LIN {X 0,Y 248.966,Z 382.302,A -85,B 0,C 180,E1 -18796.531,E2 -18796.531} C_VEL
LIN {X 0,Y 248.134,Z 387.569,A -85,B 0,C 180,E1 -18798.563,E2 -18798.563} C_VEL
LIN {X 0,Y 247.427,Z 392.65,A -85,B 0,C 180,E1 -18801.011,E2 -18801.011} C_VEL
LIN {X 0,Y 247.018,Z 396.559,A -85,B 0,C 180,E1 -18803.464,E2 -18803.464} C_VEL
LIN {X 0,Y 246.885,Z 398.563,A -85,B 0,C 180,E1 -18805.099,E2 -18805.099} C_VEL
LIN {X 0,Y 246.837,Z 400.141,A -85,B 0,C 180,E1 -18806.734,E2 -18806.734} C_VEL
LIN {X 0,Y 246.861,Z 401.271,A -85,B 0,C 180,E1 -18808.367,E2 -18808.367} C_VEL
LIN {X 0,Y 246.921,Z 401.968,A -85,B 0,C 180,E1 -18809.998,E2 -18809.998} C_VEL
LIN {X 0,Y 246.86,Z 402.267,A -85,B 0,C 180,E1 -18811.63,E2 -18811.63} C_VEL
LIN {X 0,Y 246.829,Z 402.176,A -85,B 0,C 180,E1 -18813.263,E2 -18813.263} C_VEL
LIN {X 0,Y 246.946,Z 401.583,A -85,B 0,C 180,E1 -18815.062,E2 -18815.062} C_VEL
LIN {X 0,Y 247.394,Z 399.421,A -85,B 0,C 180,E1 -18818.164,E2 -18818.164} C_VEL
LIN {X 0,Y 248.119,Z 396.646,A -85,B 0,C 180,E1 -18820.608,E2 -18820.608} C_VEL
LIN {X 0,Y 249.172,Z 392.86,A -85,B 0,C 180,E1 -18823.039,E2 -18823.039} C_VEL
LIN {X 0,Y 250.607,Z 387.967,A -85,B 0,C 180,E1 -18825.449,E2 -18825.449} C_VEL
LIN {X 0,Y 252.683,Z 381.811,A -85,B 0,C 180,E1 -18827.813,E2 -18827.813} C_VEL
LIN {X 0,Y 254.54,Z 374.922,A -85,B 0,C 180,E1 -18829.967,E2 -18829.967} C_VEL
LIN {X 0,Y 257.036,Z 366.458,A -85,B 0,C 180,E1 -18832.081,E2 -18832.081} C_VEL
LIN {X 0,Y 259.876,Z 355.993,A -85,B 0,C 180,E1 -18834.142,E2 -18834.142} C_VEL
LIN {X 0,Y 262.461,Z 345.405,A -85,B 0,C 180,E1 -18835.791,E2 -18835.791} C_VEL
LIN {X 0,Y 264.624,Z 335.228,A -85,B 0,C 180,E1 -18837.051,E2 -18837.051} C_VEL
LIN {X 0,Y 266.772,Z 323.194,A -85,B 0,C 180,E1 -18838.198,E2 -18838.198} C_VEL
LIN {X 0,Y 268.614,Z 310.075,A -85,B 0,C 180,E1 -18839.108,E2 -18839.108} C_VEL
LIN {X 0,Y 269.834,Z 297.199,A -85,B 0,C 180,E1 -18839.712,E2 -18839.712} C_VEL
LIN {X 0,Y 272.721,Z 239.475,A -85,B 0,C 180,E1 -18841.391,E2 -18841.391} C_VEL
LIN {X 0,Y 270.833,Z 226.518,A -85,B 0,C 180,E1 -18842.191,E2 -18842.191} C_VEL
LIN {X 0,Y 264.34,Z 211.708,A -85,B 0,C 180,E1 -18843.938,E2 -18843.938} C_VEL
LIN {X 0,Y 257.567,Z 198.837,A -85,B 0,C 180,E1 -18845.846,E2 -18845.846} C_VEL
LIN {X 0,Y 254.159,Z 193.208,A -85,B 0,C 180,E1 -18846.839,E2 -18846.839} C_VEL
LIN {X 0,Y 252.073,Z 189.302,A -85,B 0,C 180,E1 -18847.575,E2 -18847.575} C_VEL
LIN {X 0,Y 250.298,Z 183.421,A -85,B 0,C 180,E1 -18850.7,E2 -18850.7} C_VEL
LIN {X 0,Y 249,Z 179.025,A -85,B 0,C 180,E1 -18853.422,E2 -18853.422} C_VEL
LIN {X 0,Y 248.987,Z 178.968,A -85,B 0,C 180,E1 -18857.356,E2 -18857.356} C_VEL
LIN {X 0,Y 249.028,Z 178.958,A -85,B 0,C 180,E1 -18862.201,E2 -18862.201} C_VEL
LIN {X 0,Y 249.035,Z 178.955,A -85,B 0,C 180,E1 -18865.637,E2 -18865.637} C_VEL
LIN {X 0,Y 248.993,Z 178.96,A -85,B 0,C 180,E1 -18869.464,E2 -18869.464} C_VEL
LIN {X 0,Y 249.026,Z 178.955,A -85,B 0,C 180,E1 -18873.156,E2 -18873.156} C_VEL
LIN {X 0,Y 249.042,Z 178.952,A -85,B 0,C 180,E1 -18876.728,E2 -18876.728} C_VEL
LIN {X 0,Y 249.038,Z 178.953,A -85,B 0,C 180,E1 -18880.205,E2 -18880.205} C_VEL
LIN {X 0,Y 249.148,Z 178.944,A -85,B 0,C 180,E1 -18883.615,E2 -18883.615} C_VEL
LIN {X 0,Y 249.177,Z 178.947,A -85,B 0,C 180,E1 -18886.959,E2 -18886.959} C_VEL
LIN {X 0,Y 249.424,Z 178.909,A -85,B 0,C 180,E1 -18891.9,E2 -18891.9} C_VEL
LIN {X 0,Y 249.261,Z 178.934,A -85,B 0,C 180,E1 -18895.147,E2 -18895.147} C_VEL
LIN {X 0,Y 249.647,Z 178.889,A -85,B 0,C 180,E1 -18898.386,E2 -18898.386} C_VEL
LIN {X 0,Y 249.65,Z 178.888,A -85,B 0,C 180,E1 -18901.612,E2 -18901.612} C_VEL
LIN {X 0,Y 249.41,Z 178.911,A -85,B 0,C 180,E1 -18906.758,E2 -18906.758} C_VEL
LIN {X 0,Y 249.322,Z 178.925,A -85,B 0,C 180,E1 -18909.737,E2 -18909.737} C_VEL
LIN {X 0,Y 249.18,Z 178.997,A -85,B 0,C 180,E1 -18913.04,E2 -18913.04} C_VEL
LIN {X 0,Y 250.685,Z 184.007,A -85,B 0,C 180,E1 -18916.071,E2 -18916.071} C_VEL
LIN {X 0,Y 251.242,Z 185.375,A -85,B 0,C 180,E1 -18916.415,E2 -18916.415} C_VEL
LIN {X 0,Y 254.874,Z 191.202,A -85,B 0,C 180,E1 -18917.515,E2 -18917.515} C_VEL
LIN {X 0,Y 259.559,Z 198.978,A -85,B 0,C 180,E1 -18918.864,E2 -18918.864} C_VEL
LIN {X 0,Y 265.571,Z 210.177,A -85,B 0,C 180,E1 -18920.512,E2 -18920.512} C_VEL
LIN {X 0,Y 271.983,Z 224.396,A -85,B 0,C 180,E1 -18922.205,E2 -18922.205} C_VEL
LIN {X 0,Y 273.287,Z 227.948,A -85,B 0,C 180,E1 -18922.557,E2 -18922.557} C_VEL
LIN {X 0,Y 269.932,Z 292.598,A -85,B 0,C 180,E1 -18924.448,E2 -18924.448} C_VEL
LIN {X 0,Y 268.574,Z 306.125,A -85,B 0,C 180,E1 -18925.136,E2 -18925.136} C_VEL
LIN {X 0,Y 266.927,Z 318.251,A -85,B 0,C 180,E1 -18926.045,E2 -18926.045} C_VEL
LIN {X 0,Y 264.797,Z 330.108,A -85,B 0,C 180,E1 -18927.242,E2 -18927.242} C_VEL
LIN {X 0,Y 262.212,Z 342.255,A -85,B 0,C 180,E1 -18928.845,E2 -18928.845} C_VEL
LIN {X 0,Y 259.534,Z 353.022,A -85,B 0,C 180,E1 -18930.689,E2 -18930.689} C_VEL
LIN {X 0,Y 256.751,Z 362.823,A -85,B 0,C 180,E1 -18932.805,E2 -18932.805} C_VEL
LIN {X 0,Y 254.434,Z 370.776,A -85,B 0,C 180,E1 -18934.981,E2 -18934.981} C_VEL
LIN {X 0,Y 252.359,Z 377.241,A -85,B 0,C 180,E1 -18937.177,E2 -18937.177} C_VEL
LIN {X 0,Y 250.679,Z 382.544,A -85,B 0,C 180,E1 -18939.432,E2 -18939.432} C_VEL
LIN {X 0,Y 249.323,Z 386.724,A -85,B 0,C 180,E1 -18941.674,E2 -18941.674} C_VEL
LIN {X 0,Y 247.949,Z 391.02,A -85,B 0,C 180,E1 -18944.881,E2 -18944.881} C_VEL
LIN {X 0,Y 247.175,Z 393.392,A -85,B 0,C 180,E1 -18947.668,E2 -18947.668} C_VEL
LIN {X 0,Y 246.682,Z 394.526,A -85,B 0,C 180,E1 -18950.284,E2 -18950.284} C_VEL
LIN {X 0,Y 246.446,Z 394.592,A -85,B 0,C 180,E1 -18953.214,E2 -18953.214} C_VEL
LIN {X 0,Y 246.423,Z 393.558,A -85,B 0,C 180,E1 -18955.799,E2 -18955.799} C_VEL
LIN {X 0,Y 246.75,Z 391.147,A -85,B 0,C 180,E1 -18958.7,E2 -18958.7} C_VEL
LIN {X 0,Y 247.237,Z 388.115,A -85,B 0,C 180,E1 -18961.105,E2 -18961.105} C_VEL
LIN {X 0,Y 247.938,Z 383.166,A -85,B 0,C 180,E1 -18963.939,E2 -18963.939} C_VEL
LIN {X 0,Y 248.979,Z 376.714,A -85,B 0,C 180,E1 -18966.725,E2 -18966.725} C_VEL
LIN {X 0,Y 250.099,Z 369.969,A -85,B 0,C 180,E1 -18969.007,E2 -18969.007} C_VEL
LIN {X 0,Y 251.742,Z 361.136,A -85,B 0,C 180,E1 -18971.381,E2 -18971.381} C_VEL
LIN {X 0,Y 253.411,Z 351.377,A -85,B 0,C 180,E1 -18973.487,E2 -18973.487} C_VEL
LIN {X 0,Y 254.989,Z 341.933,A -85,B 0,C 180,E1 -18975.121,E2 -18975.121} C_VEL
LIN {X 0,Y 256.718,Z 330.09,A -85,B 0,C 180,E1 -18976.747,E2 -18976.747} C_VEL
LIN {X 0,Y 258.175,Z 318.291,A -85,B 0,C 180,E1 -18978.005,E2 -18978.005} C_VEL
LIN {X 0,Y 259.364,Z 305.706,A -85,B 0,C 180,E1 -18979.002,E2 -18979.002} C_VEL
LIN {X 0,Y 260.44,Z 291.931,A -85,B 0,C 180,E1 -18979.728,E2 -18979.728} C_VEL
LIN {X 0,Y 262.818,Z 221.817,A -85,B 0,C 180,E1 -18981.827,E2 -18981.827} C_VEL
LIN {X 0,Y 261.057,Z 212.59,A -85,B 0,C 180,E1 -18982.293,E2 -18982.293} C_VEL
LIN {X 0,Y 252.445,Z 188.907,A -85,B 0,C 180,E1 -18983.934,E2 -18983.934} C_VEL
LIN {X 0,Y 250.325,Z 183.576,A -85,B 0,C 180,E1 -18984.413,E2 -18984.413} C_VEL
LIN {X 0,Y 249.405,Z 178.982,A -85,B 0,C 180,E1 -18986.367,E2 -18986.367} C_VEL
LIN {X 0,Y 249.674,Z 178.884,A -85,B 0,C 180,E1 -18988.389,E2 -18988.389} C_VEL
LIN {X 0,Y 249.673,Z 178.882,A -85,B 0,C 180,E1 -18991.615,E2 -18991.615} C_VEL
LIN {X 0,Y 249.445,Z 178.912,A -85,B 0,C 180,E1 -18996.472,E2 -18996.472} C_VEL
LIN {X 0,Y 249.341,Z 178.927,A -85,B 0,C 180,E1 -18999.738,E2 -18999.738} C_VEL
LIN {X 0,Y 249.204,Z 178.941,A -85,B 0,C 180,E1 -19004.705,E2 -19004.705} C_VEL
LIN {X 0,Y 249.139,Z 178.942,A -85,B 0,C 180,E1 -19008.079,E2 -19008.079} C_VEL
LIN {X 0,Y 249.087,Z 178.959,A -85,B 0,C 180,E1 -19011.52,E2 -19011.52} C_VEL
LIN {X 0,Y 249.13,Z 178.939,A -85,B 0,C 180,E1 -19015.483,E2 -19015.483} C_VEL
LIN {X 0,Y 249.073,Z 178.955,A -85,B 0,C 180,E1 -19018.99,E2 -19018.99} C_VEL
LIN {X 0,Y 249.031,Z 178.963,A -85,B 0,C 180,E1 -19022.427,E2 -19022.427} C_VEL
LIN {X 0,Y 249.03,Z 178.944,A -85,B 0,C 180,E1 -19026.347,E2 -19026.347} C_VEL
LIN {X 0,Y 249.007,Z 178.965,A -85,B 0,C 180,E1 -19030.479,E2 -19030.479} C_VEL
LIN {X 0,Y 249.008,Z 178.96,A -85,B 0,C 180,E1 -19034.879,E2 -19034.879} C_VEL
LIN {X 0,Y 249.019,Z 178.943,A -85,B 0,C 180,E1 -19037.365,E2 -19037.365} C_VEL
LIN {X 0,Y 249.042,Z 178.955,A -85,B 0,C 180,E1 -19042.202,E2 -19042.202} C_VEL
LIN {X 0,Y 249.044,Z 178.961,A -85,B 0,C 180,E1 -19045.64,E2 -19045.64} C_VEL
LIN {X 0,Y 249.003,Z 178.959,A -85,B 0,C 180,E1 -19049.467,E2 -19049.467} C_VEL
LIN {X 0,Y 249.037,Z 178.962,A -85,B 0,C 180,E1 -19053.159,E2 -19053.159} C_VEL
LIN {X 0,Y 249.059,Z 178.953,A -85,B 0,C 180,E1 -19056.731,E2 -19056.731} C_VEL
LIN {X 0,Y 249.112,Z 178.955,A -85,B 0,C 180,E1 -19060.212,E2 -19060.212} C_VEL
LIN {X 0,Y 249.226,Z 178.935,A -85,B 0,C 180,E1 -19063.622,E2 -19063.622} C_VEL
LIN {X 0,Y 249.246,Z 178.936,A -85,B 0,C 180,E1 -19068.617,E2 -19068.617} C_VEL
LIN {X 0,Y 249.42,Z 178.91,A -85,B 0,C 180,E1 -19071.902,E2 -19071.902} C_VEL
LIN {X 0,Y 249.264,Z 178.933,A -85,B 0,C 180,E1 -19075.149,E2 -19075.149} C_VEL
LIN {X 0,Y 249.663,Z 178.881,A -85,B 0,C 180,E1 -19078.388,E2 -19078.388} C_VEL
LIN {X 0,Y 249.661,Z 178.865,A -85,B 0,C 180,E1 -19081.614,E2 -19081.614} C_VEL
LIN {X 0,Y 249.431,Z 178.906,A -85,B 0,C 180,E1 -19086.472,E2 -19086.472} C_VEL
LIN {X 0,Y 249.347,Z 178.926,A -85,B 0,C 180,E1 -19089.737,E2 -19089.737} C_VEL
LIN {X 0,Y 249.19,Z 178.939,A -85,B 0,C 180,E1 -19092.163,E2 -19092.163} C_VEL
LIN {X 0,Y 248.494,Z 179.024,A -85,B 0,C 180,E1 -19093.513,E2 -19093.513} C_VEL
LIN {X 0,Y 245.601,Z 179.381,A -85,B 0,C 180,E1 -19095.712,E2 -19095.712} C_VEL
LIN {X 0,Y 243.146,Z 179.686,A -85,B 0,C 180,E1 -19097.504,E2 -19097.504} C_VEL
LIN {X 0,Y 242.078,Z 179.824,A -85,B 0,C 180,E1 -19098.895,E2 -19098.895} C_VEL
LIN {X 0,Y 241.982,Z 179.833,A -85,B 0,C 180,E1 -19099.366,E2 -19099.366} C_VEL
LIN {X 0,Y 241.977,Z 179.841,A -85,B 0,C 180,E1 -19102.184,E2 -19102.184} C_VEL
LIN {X 0,Y 241.991,Z 179.824,A -85,B 0,C 180,E1 -19105.827,E2 -19105.827} C_VEL
LIN {X 0,Y 241.972,Z 179.844,A -85,B 0,C 180,E1 -19109.589,E2 -19109.589} C_VEL
LIN {X 0,Y 241.984,Z 179.83,A -85,B 0,C 180,E1 -19113.493,E2 -19113.493} C_VEL
LIN {X 0,Y 241.988,Z 179.841,A -85,B 0,C 180,E1 -19117.583,E2 -19117.583} C_VEL
LIN {X 0,Y 241.912,Z 179.85,A -85,B 0,C 180,E1 -19121.929,E2 -19121.929} C_VEL
LIN {X 0,Y 241.904,Z 179.851,A -85,B 0,C 180,E1 -19126.58,E2 -19126.58} C_VEL
LIN {X 0,Y 241.979,Z 179.842,A -85,B 0,C 180,E1 -19131.646,E2 -19131.646} C_VEL
LIN {X 0,Y 242.01,Z 179.971,A -85,B 0,C 180,E1 -19134.56,E2 -19134.56} C_VEL
LIN {X 0,Y 243.636,Z 187.404,A -85,B 0,C 180,E1 -19137.746,E2 -19137.746} C_VEL
LIN {X 0,Y 244.356,Z 190.774,A -85,B 0,C 180,E1 -19139.014,E2 -19139.014} C_VEL
LIN {X 0,Y 251.771,Z 210.686,A -85,B 0,C 180,E1 -19140.527,E2 -19140.527} C_VEL
LIN {X 0,Y 252.89,Z 215.079,A -85,B 0,C 180,E1 -19140.788,E2 -19140.788} C_VEL
LIN {X 0,Y 256.022,Z 236.939,A -85,B 0,C 180,E1 -19141.825,E2 -19141.825} C_VEL
LIN {X 0,Y 253.703,Z 299.6,A -85,B 0,C 180,E1 -19143.744,E2 -19143.744} C_VEL
LIN {X 0,Y 252.659,Z 312.872,A -85,B 0,C 180,E1 -19144.458,E2 -19144.458} C_VEL
LIN {X 0,Y 251.367,Z 325.12,A -85,B 0,C 180,E1 -19145.423,E2 -19145.423} C_VEL
LIN {X 0,Y 249.605,Z 337.75,A -85,B 0,C 180,E1 -19146.783,E2 -19146.783} C_VEL
LIN {X 0,Y 247.858,Z 349.062,A -85,B 0,C 180,E1 -19148.368,E2 -19148.368} C_VEL
LIN {X 0,Y 246.028,Z 359.736,A -85,B 0,C 180,E1 -19150.275,E2 -19150.275} C_VEL
LIN {X 0,Y 244.414,Z 369.293,A -85,B 0,C 180,E1 -19152.425,E2 -19152.425} C_VEL
LIN {X 0,Y 242.72,Z 378.086,A -85,B 0,C 180,E1 -19154.893,E2 -19154.893} C_VEL
LIN {X 0,Y 241.446,Z 385.083,A -85,B 0,C 180,E1 -19157.389,E2 -19157.389} C_VEL
LIN {X 0,Y 240.614,Z 390.675,A -85,B 0,C 180,E1 -19159.905,E2 -19159.905} C_VEL
LIN {X 0,Y 240.056,Z 395.032,A -85,B 0,C 180,E1 -19162.428,E2 -19162.428} C_VEL
LIN {X 0,Y 239.772,Z 398.622,A -85,B 0,C 180,E1 -19165.269,E2 -19165.269} C_VEL
LIN {X 0,Y 239.775,Z 401.079,A -85,B 0,C 180,E1 -19168.319,E2 -19168.319} C_VEL
LIN {X 0,Y 239.832,Z 401.81,A -85,B 0,C 180,E1 -19169.998,E2 -19169.998} C_VEL
LIN {X 0,Y 239.774,Z 402.14,A -85,B 0,C 180,E1 -19171.678,E2 -19171.678} C_VEL
LIN {X 0,Y 239.846,Z 401.628,A -85,B 0,C 180,E1 -19175.041,E2 -19175.041} C_VEL
LIN {X 0,Y 240.036,Z 400.739,A -85,B 0,C 180,E1 -19176.724,E2 -19176.724} C_VEL
LIN {X 0,Y 240.814,Z 397.763,A -85,B 0,C 180,E1 -19180.083,E2 -19180.083} C_VEL
LIN {X 0,Y 241.82,Z 394.384,A -85,B 0,C 180,E1 -19182.588,E2 -19182.588} C_VEL
LIN {X 0,Y 243.15,Z 389.945,A -85,B 0,C 180,E1 -19185.076,E2 -19185.076} C_VEL
LIN {X 0,Y 245.541,Z 383.27,A -85,B 0,C 180,E1 -19187.918,E2 -19187.918} C_VEL
LIN {X 0,Y 247.416,Z 377.362,A -85,B 0,C 180,E1 -19189.928,E2 -19189.928} C_VEL
LIN {X 0,Y 249.531,Z 370.286,A -85,B 0,C 180,E1 -19191.91,E2 -19191.91} C_VEL
LIN {X 0,Y 252.064,Z 361.749,A -85,B 0,C 180,E1 -19193.844,E2 -19193.844} C_VEL
LIN {X 0,Y 254.899,Z 351.279,A -85,B 0,C 180,E1 -19195.736,E2 -19195.736} C_VEL
LIN {X 0,Y 257.702,Z 339.544,A -85,B 0,C 180,E1 -19197.398,E2 -19197.398} C_VEL
LIN {X 0,Y 260.125,Z 327.788,A -85,B 0,C 180,E1 -19198.655,E2 -19198.655} C_VEL
LIN {X 0,Y 262.049,Z 315.767,A -85,B 0,C 180,E1 -19199.633,E2 -19199.633} C_VEL
LIN {X 0,Y 263.622,Z 302.876,A -85,B 0,C 180,E1 -19200.375,E2 -19200.375} C_VEL
LIN {X 0,Y 264.711,Z 288.127,A -85,B 0,C 180,E1 -19200.888,E2 -19200.888} C_VEL
LIN {X 0,Y 267.122,Z 240.371,A -85,B 0,C 180,E1 -19202.305,E2 -19202.305} C_VEL
LIN {X 0,Y 265.472,Z 229.249,A -85,B 0,C 180,E1 -19203.032,E2 -19203.032} C_VEL
LIN {X 0,Y 259.41,Z 215.401,A -85,B 0,C 180,E1 -19204.745,E2 -19204.745} C_VEL
LIN {X 0,Y 253.533,Z 203.887,A -85,B 0,C 180,E1 -19206.496,E2 -19206.496} C_VEL
LIN {X 0,Y 247.411,Z 193.745,A -85,B 0,C 180,E1 -19208.387,E2 -19208.387} C_VEL
LIN {X 0,Y 244.751,Z 189.183,A -85,B 0,C 180,E1 -19209.374,E2 -19209.374} C_VEL
LIN {X 0,Y 242.894,Z 183.212,A -85,B 0,C 180,E1 -19212.841,E2 -19212.841} C_VEL
LIN {X 0,Y 241.914,Z 179.884,A -85,B 0,C 180,E1 -19215.144,E2 -19215.144} C_VEL
LIN {X 0,Y 241.905,Z 179.847,A -85,B 0,C 180,E1 -19219.054,E2 -19219.054} C_VEL
LIN {X 0,Y 241.974,Z 179.836,A -85,B 0,C 180,E1 -19222.414,E2 -19222.414} C_VEL
LIN {X 0,Y 241.972,Z 179.838,A -85,B 0,C 180,E1 -19226.505,E2 -19226.505} C_VEL
LIN {X 0,Y 241.968,Z 179.844,A -85,B 0,C 180,E1 -19230.611,E2 -19230.611} C_VEL
LIN {X 0,Y 242.024,Z 179.835,A -85,B 0,C 180,E1 -19234.177,E2 -19234.177} C_VEL
LIN {X 0,Y 241.983,Z 179.841,A -85,B 0,C 180,E1 -19238.332,E2 -19238.332} C_VEL
LIN {X 0,Y 242.104,Z 179.824,A -85,B 0,C 180,E1 -19243.317,E2 -19243.317} C_VEL
LIN {X 0,Y 242.151,Z 179.812,A -85,B 0,C 180,E1 -19248.277,E2 -19248.277} C_VEL
LIN {X 0,Y 242.373,Z 179.789,A -85,B 0,C 180,E1 -19251.663,E2 -19251.663} C_VEL
LIN {X 0,Y 242.395,Z 179.781,A -85,B 0,C 180,E1 -19253.339,E2 -19253.339} C_VEL
LIN {X 0,Y 242.607,Z 179.765,A -85,B 0,C 180,E1 -19258.339,E2 -19258.339} C_VEL
LIN {X 0,Y 242.609,Z 179.765,A -85,B 0,C 180,E1 -19261.659,E2 -19261.659} C_VEL
LIN {X 0,Y 242.39,Z 179.786,A -85,B 0,C 180,E1 -19266.731,E2 -19266.731} C_VEL
LIN {X 0,Y 242.25,Z 179.808,A -85,B 0,C 180,E1 -19270.024,E2 -19270.024} C_VEL
LIN {X 0,Y 242.187,Z 179.963,A -85,B 0,C 180,E1 -19271.507,E2 -19271.507} C_VEL
LIN {X 0,Y 243.558,Z 184.504,A -85,B 0,C 180,E1 -19274.357,E2 -19274.357} C_VEL
LIN {X 0,Y 246.527,Z 189.136,A -85,B 0,C 180,E1 -19275.448,E2 -19275.448} C_VEL
LIN {X 0,Y 253.165,Z 199.962,A -85,B 0,C 180,E1 -19277.531,E2 -19277.531} C_VEL
LIN {X 0,Y 260.169,Z 212.884,A -85,B 0,C 180,E1 -19279.585,E2 -19279.585} C_VEL
LIN {X 0,Y 266,Z 225.762,A -85,B 0,C 180,E1 -19281.205,E2 -19281.205} C_VEL
LIN {X 0,Y 267.675,Z 229.833,A -85,B 0,C 180,E1 -19281.664,E2 -19281.664} C_VEL
LIN {X 0,Y 264.236,Z 292.445,A -85,B 0,C 180,E1 -19283.535,E2 -19283.535} C_VEL
LIN {X 0,Y 262.797,Z 306.223,A -85,B 0,C 180,E1 -19284.246,E2 -19284.246} C_VEL
LIN {X 0,Y 260.891,Z 319.326,A -85,B 0,C 180,E1 -19285.26,E2 -19285.26} C_VEL
LIN {X 0,Y 258.537,Z 331.741,A -85,B 0,C 180,E1 -19286.568,E2 -19286.568} C_VEL
LIN {X 0,Y 255.948,Z 343.152,A -85,B 0,C 180,E1 -19288.139,E2 -19288.139} C_VEL
LIN {X 0,Y 253.205,Z 353.544,A -85,B 0,C 180,E1 -19289.973,E2 -19289.973} C_VEL
LIN {X 0,Y 250.587,Z 362.306,A -85,B 0,C 180,E1 -19291.898,E2 -19291.898} C_VEL
LIN {X 0,Y 248.165,Z 370.229,A -85,B 0,C 180,E1 -19294.076,E2 -19294.076} C_VEL
LIN {X 0,Y 245.558,Z 377.876,A -85,B 0,C 180,E1 -19296.743,E2 -19296.743} C_VEL
LIN {X 0,Y 243.545,Z 383.746,A -85,B 0,C 180,E1 -19299.408,E2 -19299.408} C_VEL
LIN {X 0,Y 242.081,Z 387.942,A -85,B 0,C 180,E1 -19301.891,E2 -19301.891} C_VEL
LIN {X 0,Y 241.018,Z 391.097,A -85,B 0,C 180,E1 -19304.412,E2 -19304.412} C_VEL
LIN {X 0,Y 240.075,Z 393.741,A -85,B 0,C 180,E1 -19307.68,E2 -19307.68} C_VEL
LIN {X 0,Y 239.641,Z 394.59,A -85,B 0,C 180,E1 -19309.823,E2 -19309.823} C_VEL
LIN {X 0,Y 239.375,Z 394.773,A -85,B 0,C 180,E1 -19312.439,E2 -19312.439} C_VEL
LIN {X 0,Y 239.303,Z 393.855,A -85,B 0,C 180,E1 -19315.316,E2 -19315.316} C_VEL
LIN {X 0,Y 239.586,Z 391.661,A -85,B 0,C 180,E1 -19318.285,E2 -19318.285} C_VEL
LIN {X 0,Y 240.199,Z 387.896,A -85,B 0,C 180,E1 -19321.373,E2 -19321.373} C_VEL
LIN {X 0,Y 240.872,Z 383.325,A -85,B 0,C 180,E1 -19324.048,E2 -19324.048} C_VEL
LIN {X 0,Y 241.95,Z 376.884,A -85,B 0,C 180,E1 -19326.915,E2 -19326.915} C_VEL
LIN {X 0,Y 243.088,Z 370.164,A -85,B 0,C 180,E1 -19329.26,E2 -19329.26} C_VEL
LIN {X 0,Y 244.707,Z 361.812,A -85,B 0,C 180,E1 -19331.586,E2 -19331.586} C_VEL
LIN {X 0,Y 246.477,Z 351.827,A -85,B 0,C 180,E1 -19333.818,E2 -19333.818} C_VEL
LIN {X 0,Y 248.289,Z 341.402,A -85,B 0,C 180,E1 -19335.662,E2 -19335.662} C_VEL
LIN {X 0,Y 250.109,Z 329.213,A -85,B 0,C 180,E1 -19337.353,E2 -19337.353} C_VEL
LIN {X 0,Y 251.546,Z 317.754,A -85,B 0,C 180,E1 -19338.583,E2 -19338.583} C_VEL
LIN {X 0,Y 252.786,Z 304.681,A -85,B 0,C 180,E1 -19339.616,E2 -19339.616} C_VEL
LIN {X 0,Y 253.893,Z 290.762,A -85,B 0,C 180,E1 -19340.341,E2 -19340.341} C_VEL
LIN {X 0,Y 256.246,Z 222.797,A -85,B 0,C 180,E1 -19342.413,E2 -19342.413} C_VEL
LIN {X 0,Y 254.735,Z 214.758,A -85,B 0,C 180,E1 -19342.828,E2 -19342.828} C_VEL
LIN {X 0,Y 246.327,Z 191.636,A -85,B 0,C 180,E1 -19344.487,E2 -19344.487} C_VEL
LIN {X 0,Y 243.215,Z 184.115,A -85,B 0,C 180,E1 -19345.133,E2 -19345.133} C_VEL
LIN {X 0,Y 242.951,Z 183.003,A -85,B 0,C 180,E1 -19345.439,E2 -19345.439} C_VEL
LIN {X 0,Y 242.41,Z 179.845,A -85,B 0,C 180,E1 -19346.886,E2 -19346.886} C_VEL
LIN {X 0,Y 242.689,Z 179.752,A -85,B 0,C 180,E1 -19350.002,E2 -19350.002} C_VEL
LIN {X 0,Y 242.633,Z 179.759,A -85,B 0,C 180,E1 -19351.662,E2 -19351.662} C_VEL
LIN {X 0,Y 242.415,Z 179.788,A -85,B 0,C 180,E1 -19356.661,E2 -19356.661} C_VEL
LIN {X 0,Y 242.265,Z 179.808,A -85,B 0,C 180,E1 -19360.025,E2 -19360.025} C_VEL
LIN {X 0,Y 242.166,Z 179.819,A -85,B 0,C 180,E1 -19365.142,E2 -19365.142} C_VEL
LIN {X 0,Y 242.073,Z 179.82,A -85,B 0,C 180,E1 -19368.626,E2 -19368.626} C_VEL
LIN {X 0,Y 242.013,Z 179.838,A -85,B 0,C 180,E1 -19372.181,E2 -19372.181} C_VEL
LIN {X 0,Y 242.067,Z 179.817,A -85,B 0,C 180,E1 -19375.84,E2 -19375.84} C_VEL
LIN {X 0,Y 242.007,Z 179.839,A -85,B 0,C 180,E1 -19379.585,E2 -19379.585} C_VEL
LIN {X 0,Y 241.981,Z 179.835,A -85,B 0,C 180,E1 -19383.494,E2 -19383.494} C_VEL
LIN {X 0,Y 241.986,Z 179.827,A -85,B 0,C 180,E1 -19387.584,E2 -19387.584} C_VEL
LIN {X 0,Y 241.94,Z 179.846,A -85,B 0,C 180,E1 -19391.923,E2 -19391.923} C_VEL
LIN {X 0,Y 241.938,Z 179.829,A -85,B 0,C 180,E1 -19396.572,E2 -19396.572} C_VEL
LIN {X 0,Y 241.957,Z 179.825,A -85,B 0,C 180,E1 -19400.282,E2 -19400.282} C_VEL
LIN {X 0,Y 241.981,Z 179.843,A -85,B 0,C 180,E1 -19404.489,E2 -19404.489} C_VEL
LIN {X 0,Y 241.954,Z 179.84,A -85,B 0,C 180,E1 -19408.478,E2 -19408.478} C_VEL
LIN {X 0,Y 241.97,Z 179.845,A -85,B 0,C 180,E1 -19412.309,E2 -19412.309} C_VEL
LIN {X 0,Y 242.028,Z 179.831,A -85,B 0,C 180,E1 -19416.014,E2 -19416.014} C_VEL
LIN {X 0,Y 242.039,Z 179.832,A -85,B 0,C 180,E1 -19419.609,E2 -19419.609} C_VEL
LIN {X 0,Y 242.167,Z 179.814,A -85,B 0,C 180,E1 -19423.279,E2 -19423.279} C_VEL
LIN {X 0,Y 242.182,Z 179.817,A -85,B 0,C 180,E1 -19428.28,E2 -19428.28} C_VEL
LIN {X 0,Y 242.374,Z 179.788,A -85,B 0,C 180,E1 -19431.665,E2 -19431.665} C_VEL
LIN {X 0,Y 242.399,Z 179.783,A -85,B 0,C 180,E1 -19433.341,E2 -19433.341} C_VEL
LIN {X 0,Y 242.622,Z 179.758,A -85,B 0,C 180,E1 -19438.341,E2 -19438.341} C_VEL
LIN {X 0,Y 242.621,Z 179.74,A -85,B 0,C 180,E1 -19441.661,E2 -19441.661} C_VEL
LIN {X 0,Y 242.404,Z 179.781,A -85,B 0,C 180,E1 -19446.66,E2 -19446.66} C_VEL
LIN {X 0,Y 242.27,Z 179.806,A -85,B 0,C 180,E1 -19450.024,E2 -19450.024} C_VEL
LIN {X 0,Y 242.125,Z 179.804,A -85,B 0,C 180,E1 -19455.144,E2 -19455.144} C_VEL
LIN {X 0,Y 241.982,Z 179.833,A -85,B 0,C 180,E1 -19459.366,E2 -19459.366} C_VEL
LIN {X 0,Y 241.308,Z 179.927,A -85,B 0,C 180,E1 -19460.754,E2 -19460.754} C_VEL
LIN {X 0,Y 238.507,Z 180.273,A -85,B 0,C 180,E1 -19463.019,E2 -19463.019} C_VEL
LIN {X 0,Y 235.282,Z 180.663,A -85,B 0,C 180,E1 -19465.812,E2 -19465.812} C_VEL
LIN {X 0,Y 234.92,Z 180.705,A -85,B 0,C 180,E1 -19466.778,E2 -19466.778} C_VEL
LIN {X 0,Y 234.903,Z 180.725,A -85,B 0,C 180,E1 -19470.573,E2 -19470.573} C_VEL
LIN {X 0,Y 234.93,Z 180.709,A -85,B 0,C 180,E1 -19474.639,E2 -19474.639} C_VEL
LIN {X 0,Y 234.917,Z 180.716,A -85,B 0,C 180,E1 -19478.935,E2 -19478.935} C_VEL
LIN {X 0,Y 234.858,Z 180.728,A -85,B 0,C 180,E1 -19483.494,E2 -19483.494} C_VEL
LIN {X 0,Y 234.856,Z 180.728,A -85,B 0,C 180,E1 -19486.505,E2 -19486.505} C_VEL
LIN {X 0,Y 234.923,Z 180.72,A -85,B 0,C 180,E1 -19491.078,E2 -19491.078} C_VEL
LIN {X 0,Y 234.94,Z 180.887,A -85,B 0,C 180,E1 -19494.03,E2 -19494.03} C_VEL
LIN {X 0,Y 236.795,Z 189.252,A -85,B 0,C 180,E1 -19497.706,E2 -19497.706} C_VEL
LIN {X 0,Y 237.088,Z 190.758,A -85,B 0,C 180,E1 -19498.19,E2 -19498.19} C_VEL
LIN {X 0,Y 243.253,Z 206.795,A -85,B 0,C 180,E1 -19499.511,E2 -19499.511} C_VEL
LIN {X 0,Y 246.356,Z 215.976,A -85,B 0,C 180,E1 -19500.162,E2 -19500.162} C_VEL
LIN {X 0,Y 249.461,Z 238.081,A -85,B 0,C 180,E1 -19501.242,E2 -19501.242} C_VEL
LIN {X 0,Y 247.076,Z 299.144,A -85,B 0,C 180,E1 -19503.155,E2 -19503.155} C_VEL
LIN {X 0,Y 245.941,Z 313.266,A -85,B 0,C 180,E1 -19503.936,E2 -19503.936} C_VEL
LIN {X 0,Y 244.619,Z 325.356,A -85,B 0,C 180,E1 -19504.926,E2 -19504.926} C_VEL
LIN {X 0,Y 242.814,Z 337.91,A -85,B 0,C 180,E1 -19506.32,E2 -19506.32} C_VEL
LIN {X 0,Y 241.009,Z 349.174,A -85,B 0,C 180,E1 -19507.947,E2 -19507.947} C_VEL
LIN {X 0,Y 239.252,Z 359.079,A -85,B 0,C 180,E1 -19509.754,E2 -19509.754} C_VEL
LIN {X 0,Y 237.614,Z 368.5,A -85,B 0,C 180,E1 -19511.905,E2 -19511.905} C_VEL
LIN {X 0,Y 235.851,Z 377.436,A -85,B 0,C 180,E1 -19514.442,E2 -19514.442} C_VEL
LIN {X 0,Y 234.46,Z 384.55,A -85,B 0,C 180,E1 -19517.006,E2 -19517.006} C_VEL
LIN {X 0,Y 233.585,Z 390.229,A -85,B 0,C 180,E1 -19519.598,E2 -19519.598} C_VEL
LIN {X 0,Y 233.01,Z 394.666,A -85,B 0,C 180,E1 -19522.198,E2 -19522.198} C_VEL
LIN {X 0,Y 232.677,Z 398.613,A -85,B 0,C 180,E1 -19525.397,E2 -19525.397} C_VEL
LIN {X 0,Y 232.672,Z 400.863,A -85,B 0,C 180,E1 -19528.267,E2 -19528.267} C_VEL
LIN {X 0,Y 232.745,Z 401.65,A -85,B 0,C 180,E1 -19529.998,E2 -19529.998} C_VEL
LIN {X 0,Y 232.67,Z 402.012,A -85,B 0,C 180,E1 -19531.729,E2 -19531.729} C_VEL
LIN {X 0,Y 232.77,Z 401.57,A -85,B 0,C 180,E1 -19535.195,E2 -19535.195} C_VEL
LIN {X 0,Y 232.982,Z 400.738,A -85,B 0,C 180,E1 -19536.928,E2 -19536.928} C_VEL
LIN {X 0,Y 233.806,Z 397.829,A -85,B 0,C 180,E1 -19540.388,E2 -19540.388} C_VEL
LIN {X 0,Y 234.877,Z 394.532,A -85,B 0,C 180,E1 -19542.966,E2 -19542.966} C_VEL
LIN {X 0,Y 236.298,Z 390.186,A -85,B 0,C 180,E1 -19545.524,E2 -19545.524} C_VEL
LIN {X 0,Y 238.819,Z 383.637,A -85,B 0,C 180,E1 -19548.44,E2 -19548.44} C_VEL
LIN {X 0,Y 240.74,Z 377.797,A -85,B 0,C 180,E1 -19550.505,E2 -19550.505} C_VEL
LIN {X 0,Y 243.473,Z 369.264,A -85,B 0,C 180,E1 -19552.933,E2 -19552.933} C_VEL
LIN {X 0,Y 246.198,Z 360.53,A -85,B 0,C 180,E1 -19554.899,E2 -19554.899} C_VEL
LIN {X 0,Y 249.195,Z 349.868,A -85,B 0,C 180,E1 -19556.821,E2 -19556.821} C_VEL
LIN {X 0,Y 251.856,Z 339.292,A -85,B 0,C 180,E1 -19558.317,E2 -19558.317} C_VEL
LIN {X 0,Y 254.353,Z 327.556,A -85,B 0,C 180,E1 -19559.595,E2 -19559.595} C_VEL
LIN {X 0,Y 256.591,Z 314.303,A -85,B 0,C 180,E1 -19560.67,E2 -19560.67} C_VEL
LIN {X 0,Y 258.138,Z 301.125,A -85,B 0,C 180,E1 -19561.404,E2 -19561.404} C_VEL
LIN {X 0,Y 259.436,Z 282.027,A -85,B 0,C 180,E1 -19562.034,E2 -19562.034} C_VEL
LIN {X 0,Y 261.613,Z 241.358,A -85,B 0,C 180,E1 -19563.257,E2 -19563.257} C_VEL
LIN {X 0,Y 260.1,Z 231.705,A -85,B 0,C 180,E1 -19563.933,E2 -19563.933} C_VEL
LIN {X 0,Y 254.564,Z 219.061,A -85,B 0,C 180,E1 -19565.596,E2 -19565.596} C_VEL
LIN {X 0,Y 249.089,Z 208.286,A -85,B 0,C 180,E1 -19567.299,E2 -19567.299} C_VEL
LIN {X 0,Y 243.374,Z 198.558,A -85,B 0,C 180,E1 -19569.187,E2 -19569.187} C_VEL
LIN {X 0,Y 240.376,Z 193.825,A -85,B 0,C 180,E1 -19570.237,E2 -19570.237} C_VEL
LIN {X 0,Y 237.566,Z 189.321,A -85,B 0,C 180,E1 -19571.329,E2 -19571.329} C_VEL
LIN {X 0,Y 236.988,Z 187.699,A -85,B 0,C 180,E1 -19572.149,E2 -19572.149} C_VEL
LIN {X 0,Y 234.972,Z 181.275,A -85,B 0,C 180,E1 -19576.533,E2 -19576.533} C_VEL
LIN {X 0,Y 234.848,Z 180.731,A -85,B 0,C 180,E1 -19577.284,E2 -19577.284} C_VEL
LIN {X 0,Y 234.911,Z 180.723,A -85,B 0,C 180,E1 -19581.076,E2 -19581.076} C_VEL
LIN {X 0,Y 234.921,Z 180.713,A -85,B 0,C 180,E1 -19585.36,E2 -19585.36} C_VEL
LIN {X 0,Y 234.89,Z 180.716,A -85,B 0,C 180,E1 -19589.425,E2 -19589.425} C_VEL
LIN {X 0,Y 234.96,Z 180.711,A -85,B 0,C 180,E1 -19593.805,E2 -19593.805} C_VEL
LIN {X 0,Y 234.956,Z 180.712,A -85,B 0,C 180,E1 -19598.006,E2 -19598.006} C_VEL
LIN {X 0,Y 235.045,Z 180.705,A -85,B 0,C 180,E1 -19603.092,E2 -19603.092} C_VEL
LIN {X 0,Y 235.084,Z 180.694,A -85,B 0,C 180,E1 -19607.92,E2 -19607.92} C_VEL
LIN {X 0,Y 235.307,Z 180.672,A -85,B 0,C 180,E1 -19611.411,E2 -19611.411} C_VEL
LIN {X 0,Y 235.346,Z 180.658,A -85,B 0,C 180,E1 -19613.139,E2 -19613.139} C_VEL
LIN {X 0,Y 235.567,Z 180.642,A -85,B 0,C 180,E1 -19618.29,E2 -19618.29} C_VEL
LIN {X 0,Y 235.568,Z 180.643,A -85,B 0,C 180,E1 -19621.709,E2 -19621.709} C_VEL
LIN {X 0,Y 235.347,Z 180.664,A -85,B 0,C 180,E1 -19626.86,E2 -19626.86} C_VEL
LIN {X 0,Y 235.288,Z 180.898,A -85,B 0,C 180,E1 -19629.717,E2 -19629.717} C_VEL
LIN {X 0,Y 236.398,Z 184.856,A -85,B 0,C 180,E1 -19632.337,E2 -19632.337} C_VEL
LIN {X 0,Y 239.346,Z 189.356,A -85,B 0,C 180,E1 -19633.526,E2 -19633.526} C_VEL
LIN {X 0,Y 243.681,Z 195.883,A -85,B 0,C 180,E1 -19635.044,E2 -19635.044} C_VEL
LIN {X 0,Y 249.372,Z 205.479,A -85,B 0,C 180,E1 -19636.923,E2 -19636.923} C_VEL
LIN {X 0,Y 255.603,Z 217.046,A -85,B 0,C 180,E1 -19638.819,E2 -19638.819} C_VEL
LIN {X 0,Y 261.095,Z 229.541,A -85,B 0,C 180,E1 -19640.451,E2 -19640.451} C_VEL
LIN {X 0,Y 262.115,Z 231.983,A -85,B 0,C 180,E1 -19640.74,E2 -19640.74} C_VEL
LIN {X 0,Y 258.653,Z 292.451,A -85,B 0,C 180,E1 -19642.577,E2 -19642.577} C_VEL
LIN {X 0,Y 257.139,Z 306.152,A -85,B 0,C 180,E1 -19643.286,E2 -19643.286} C_VEL
LIN {X 0,Y 255.275,Z 318.822,A -85,B 0,C 180,E1 -19644.276,E2 -19644.276} C_VEL
LIN {X 0,Y 252.776,Z 331.342,A -85,B 0,C 180,E1 -19645.601,E2 -19645.601} C_VEL
LIN {X 0,Y 250.311,Z 341.886,A -85,B 0,C 180,E1 -19647.054,E2 -19647.054} C_VEL
LIN {X 0,Y 247.429,Z 352.344,A -85,B 0,C 180,E1 -19648.872,E2 -19648.872} C_VEL
LIN {X 0,Y 244.475,Z 361.92,A -85,B 0,C 180,E1 -19650.981,E2 -19650.981} C_VEL
LIN {X 0,Y 241.841,Z 370.063,A -85,B 0,C 180,E1 -19653.243,E2 -19653.243} C_VEL
LIN {X 0,Y 239.005,Z 377.91,A -85,B 0,C 180,E1 -19656.022,E2 -19656.022} C_VEL
LIN {X 0,Y 237.056,Z 383.319,A -85,B 0,C 180,E1 -19658.504,E2 -19658.504} C_VEL
LIN {X 0,Y 235.081,Z 388.482,A -85,B 0,C 180,E1 -19661.638,E2 -19661.638} C_VEL
LIN {X 0,Y 234.096,Z 391.173,A -85,B 0,C 180,E1 -19663.906,E2 -19663.906} C_VEL
LIN {X 0,Y 233.333,Z 393.207,A -85,B 0,C 180,E1 -19666.292,E2 -19666.292} C_VEL
LIN {X 0,Y 232.688,Z 394.574,A -85,B 0,C 180,E1 -19669.032,E2 -19669.032} C_VEL
LIN {X 0,Y 232.308,Z 394.924,A -85,B 0,C 180,E1 -19671.865,E2 -19671.865} C_VEL
LIN {X 0,Y 232.187,Z 394.105,A -85,B 0,C 180,E1 -19674.896,E2 -19674.896} C_VEL
LIN {X 0,Y 232.413,Z 392.107,A -85,B 0,C 180,E1 -19677.853,E2 -19677.853} C_VEL
LIN {X 0,Y 233.054,Z 388.4,A -85,B 0,C 180,E1 -19681.154,E2 -19681.154} C_VEL
LIN {X 0,Y 233.854,Z 383.075,A -85,B 0,C 180,E1 -19684.366,E2 -19684.366} C_VEL
LIN {X 0,Y 234.899,Z 377.03,A -85,B 0,C 180,E1 -19687.113,E2 -19687.113} C_VEL
LIN {X 0,Y 236.092,Z 370.312,A -85,B 0,C 180,E1 -19689.529,E2 -19689.529} C_VEL
LIN {X 0,Y 237.771,Z 361.932,A -85,B 0,C 180,E1 -19691.929,E2 -19691.929} C_VEL
LIN {X 0,Y 239.412,Z 352.882,A -85,B 0,C 180,E1 -19694.028,E2 -19694.028} C_VEL
LIN {X 0,Y 241.221,Z 342.97,A -85,B 0,C 180,E1 -19695.879,E2 -19695.879} C_VEL
LIN {X 0,Y 242.892,Z 332.355,A -85,B 0,C 180,E1 -19697.469,E2 -19697.469} C_VEL
LIN {X 0,Y 244.632,Z 319.717,A -85,B 0,C 180,E1 -19698.925,E2 -19698.925} C_VEL
LIN {X 0,Y 245.952,Z 306.952,A -85,B 0,C 180,E1 -19700.026,E2 -19700.026} C_VEL
LIN {X 0,Y 247.051,Z 293.627,A -85,B 0,C 180,E1 -19700.794,E2 -19700.794} C_VEL
LIN {X 0,Y 247.998,Z 272.807,A -85,B 0,C 180,E1 -19701.497,E2 -19701.497} C_VEL
LIN {X 0,Y 249.721,Z 223.936,A -85,B 0,C 180,E1 -19703.007,E2 -19703.007} C_VEL
LIN {X 0,Y 248.485,Z 217.167,A -85,B 0,C 180,E1 -19703.365,E2 -19703.365} C_VEL
LIN {X 0,Y 240.43,Z 194.935,A -85,B 0,C 180,E1 -19705.013,E2 -19705.013} C_VEL
LIN {X 0,Y 235.982,Z 184.077,A -85,B 0,C 180,E1 -19705.97,E2 -19705.97} C_VEL
LIN {X 0,Y 235.448,Z 180.977,A -85,B 0,C 180,E1 -19707.222,E2 -19707.222} C_VEL
LIN {X 0,Y 235.516,Z 180.649,A -85,B 0,C 180,E1 -19707.864,E2 -19707.864} C_VEL
LIN {X 0,Y 235.653,Z 180.628,A -85,B 0,C 180,E1 -19710.002,E2 -19710.002} C_VEL
LIN {X 0,Y 235.593,Z 180.636,A -85,B 0,C 180,E1 -19711.711,E2 -19711.711} C_VEL
LIN {X 0,Y 235.366,Z 180.666,A -85,B 0,C 180,E1 -19716.861,E2 -19716.861} C_VEL
LIN {X 0,Y 235.211,Z 180.686,A -85,B 0,C 180,E1 -19720.329,E2 -19720.329} C_VEL
LIN {X 0,Y 235.113,Z 180.7,A -85,B 0,C 180,E1 -19725.608,E2 -19725.608} C_VEL
LIN {X 0,Y 235.009,Z 180.699,A -85,B 0,C 180,E1 -19729.207,E2 -19729.207} C_VEL
LIN {X 0,Y 234.961,Z 180.718,A -85,B 0,C 180,E1 -19732.884,E2 -19732.884} C_VEL
LIN {X 0,Y 234.968,Z 180.699,A -85,B 0,C 180,E1 -19736.659,E2 -19736.659} C_VEL
LIN {X 0,Y 234.923,Z 180.721,A -85,B 0,C 180,E1 -19740.571,E2 -19740.571} C_VEL
LIN {X 0,Y 234.927,Z 180.706,A -85,B 0,C 180,E1 -19744.64,E2 -19744.64} C_VEL
LIN {X 0,Y 234.943,Z 180.71,A -85,B 0,C 180,E1 -19748.946,E2 -19748.946} C_VEL
LIN {X 0,Y 234.891,Z 180.722,A -85,B 0,C 180,E1 -19753.487,E2 -19753.487} C_VEL
LIN {X 0,Y 234.891,Z 180.705,A -85,B 0,C 180,E1 -19756.516,E2 -19756.516} C_VEL
LIN {X 0,Y 234.919,Z 180.708,A -85,B 0,C 180,E1 -19761.08,E2 -19761.08} C_VEL
LIN {X 0,Y 234.927,Z 180.72,A -85,B 0,C 180,E1 -19765.362,E2 -19765.362} C_VEL
LIN {X 0,Y 234.901,Z 180.715,A -85,B 0,C 180,E1 -19769.429,E2 -19769.429} C_VEL
LIN {X 0,Y 234.971,Z 180.715,A -85,B 0,C 180,E1 -19773.808,E2 -19773.808} C_VEL
LIN {X 0,Y 235.001,Z 180.709,A -85,B 0,C 180,E1 -19778.97,E2 -19778.97} C_VEL
LIN {X 0,Y 235.099,Z 180.694,A -85,B 0,C 180,E1 -19783.061,E2 -19783.061} C_VEL
LIN {X 0,Y 235.116,Z 180.697,A -85,B 0,C 180,E1 -19787.923,E2 -19787.923} C_VEL
LIN {X 0,Y 235.314,Z 180.668,A -85,B 0,C 180,E1 -19791.413,E2 -19791.413} C_VEL
LIN {X 0,Y 235.35,Z 180.66,A -85,B 0,C 180,E1 -19793.141,E2 -19793.141} C_VEL
LIN {X 0,Y 235.581,Z 180.635,A -85,B 0,C 180,E1 -19798.291,E2 -19798.291} C_VEL
LIN {X 0,Y 235.58,Z 180.615,A -85,B 0,C 180,E1 -19801.71,E2 -19801.71} C_VEL
LIN {X 0,Y 235.356,Z 180.658,A -85,B 0,C 180,E1 -19806.861,E2 -19806.861} C_VEL
LIN {X 0,Y 235.216,Z 180.684,A -85,B 0,C 180,E1 -19810.328,E2 -19810.328} C_VEL
LIN {X 0,Y 235.074,Z 180.679,A -85,B 0,C 180,E1 -19815.61,E2 -19815.61} C_VEL
LIN {X 0,Y 234.957,Z 180.712,A -85,B 0,C 180,E1 -19819.338,E2 -19819.338} C_VEL
LIN {X 0,Y 234.913,Z 180.722,A -85,B 0,C 180,E1 -19822.889,E2 -19822.889} C_VEL
LIN {X 0,Y 234.92,Z 180.705,A -85,B 0,C 180,E1 -19826.778,E2 -19826.778} C_VEL
LIN {X 0,Y 234.193,Z 180.808,A -85,B 0,C 180,E1 -19828.209,E2 -19828.209} C_VEL
LIN {X 0,Y 231.352,Z 181.167,A -85,B 0,C 180,E1 -19830.546,E2 -19830.546} C_VEL
LIN {X 0,Y 228.969,Z 181.457,A -85,B 0,C 180,E1 -19832.45,E2 -19832.45} C_VEL
LIN {X 0,Y 227.935,Z 181.577,A -85,B 0,C 180,E1 -19833.927,E2 -19833.927} C_VEL
LIN {X 0,Y 227.842,Z 181.589,A -85,B 0,C 180,E1 -19834.428,E2 -19834.428} C_VEL
LIN {X 0,Y 227.845,Z 181.602,A -85,B 0,C 180,E1 -19838.092,E2 -19838.092} C_VEL
LIN {X 0,Y 227.79,Z 181.612,A -85,B 0,C 180,E1 -19842.748,E2 -19842.748} C_VEL
LIN {X 0,Y 227.814,Z 181.6,A -85,B 0,C 180,E1 -19845.199,E2 -19845.199} C_VEL
LIN {X 0,Y 227.802,Z 181.61,A -85,B 0,C 180,E1 -19849.617,E2 -19849.617} C_VEL
LIN {X 0,Y 227.894,Z 181.779,A -85,B 0,C 180,E1 -19853.466,E2 -19853.466} C_VEL
LIN {X 0,Y 229.8,Z 190.322,A -85,B 0,C 180,E1 -19857.275,E2 -19857.275} C_VEL
LIN {X 0,Y 232.64,Z 197.598,A -85,B 0,C 180,E1 -19857.97,E2 -19857.97} C_VEL
LIN {X 0,Y 239.838,Z 217.021,A -85,B 0,C 180,E1 -19859.509,E2 -19859.509} C_VEL
LIN {X 0,Y 242.918,Z 238.705,A -85,B 0,C 180,E1 -19860.611,E2 -19860.611} C_VEL
LIN {X 0,Y 240.505,Z 298.706,A -85,B 0,C 180,E1 -19862.537,E2 -19862.537} C_VEL
LIN {X 0,Y 239.37,Z 312.163,A -85,B 0,C 180,E1 -19863.282,E2 -19863.282} C_VEL
LIN {X 0,Y 238.023,Z 324.554,A -85,B 0,C 180,E1 -19864.298,E2 -19864.298} C_VEL
LIN {X 0,Y 236.296,Z 336.484,A -85,B 0,C 180,E1 -19865.625,E2 -19865.625} C_VEL
LIN {X 0,Y 234.585,Z 346.672,A -85,B 0,C 180,E1 -19867.077,E2 -19867.077} C_VEL
LIN {X 0,Y 232.713,Z 357.3,A -85,B 0,C 180,E1 -19868.983,E2 -19868.983} C_VEL
LIN {X 0,Y 231.096,Z 365.989,A -85,B 0,C 180,E1 -19870.916,E2 -19870.916} C_VEL
LIN {X 0,Y 229.499,Z 373.982,A -85,B 0,C 180,E1 -19873.085,E2 -19873.085} C_VEL
LIN {X 0,Y 227.932,Z 381.756,A -85,B 0,C 180,E1 -19875.718,E2 -19875.718} C_VEL
LIN {X 0,Y 226.874,Z 387.992,A -85,B 0,C 180,E1 -19878.382,E2 -19878.382} C_VEL
LIN {X 0,Y 226.143,Z 392.914,A -85,B 0,C 180,E1 -19881.059,E2 -19881.059} C_VEL
LIN {X 0,Y 225.706,Z 396.671,A -85,B 0,C 180,E1 -19883.742,E2 -19883.742} C_VEL
LIN {X 0,Y 225.574,Z 399.374,A -85,B 0,C 180,E1 -19886.426,E2 -19886.426} C_VEL
LIN {X 0,Y 225.572,Z 400.637,A -85,B 0,C 180,E1 -19888.213,E2 -19888.213} C_VEL
LIN {X 0,Y 225.659,Z 401.486,A -85,B 0,C 180,E1 -19889.998,E2 -19889.998} C_VEL
LIN {X 0,Y 225.571,Z 401.884,A -85,B 0,C 180,E1 -19891.784,E2 -19891.784} C_VEL
LIN {X 0,Y 225.694,Z 401.508,A -85,B 0,C 180,E1 -19895.358,E2 -19895.358} C_VEL
LIN {X 0,Y 225.923,Z 400.738,A -85,B 0,C 180,E1 -19897.146,E2 -19897.146} C_VEL
LIN {X 0,Y 226.814,Z 397.917,A -85,B 0,C 180,E1 -19900.712,E2 -19900.712} C_VEL
LIN {X 0,Y 227.949,Z 394.696,A -85,B 0,C 180,E1 -19903.368,E2 -19903.368} C_VEL
LIN {X 0,Y 229.468,Z 390.429,A -85,B 0,C 180,E1 -19905.998,E2 -19905.998} C_VEL
LIN {X 0,Y 232.121,Z 383.973,A -85,B 0,C 180,E1 -19908.992,E2 -19908.992} C_VEL
LIN {X 0,Y 234.294,Z 377.449,A -85,B 0,C 180,E1 -19911.39,E2 -19911.39} C_VEL
LIN {X 0,Y 236.999,Z 369.894,A -85,B 0,C 180,E1 -19913.597,E2 -19913.597} C_VEL
LIN {X 0,Y 239.825,Z 361.347,A -85,B 0,C 180,E1 -19915.608,E2 -19915.608} C_VEL
LIN {X 0,Y 242.943,Z 350.883,A -85,B 0,C 180,E1 -19917.569,E2 -19917.569} C_VEL
LIN {X 0,Y 246.055,Z 339.137,A -85,B 0,C 180,E1 -19919.281,E2 -19919.281} C_VEL
LIN {X 0,Y 248.682,Z 327.381,A -85,B 0,C 180,E1 -19920.575,E2 -19920.575} C_VEL
LIN {X 0,Y 251.005,Z 314.115,A -85,B 0,C 180,E1 -19921.665,E2 -19921.665} C_VEL
LIN {X 0,Y 252.639,Z 300.743,A -85,B 0,C 180,E1 -19922.413,E2 -19922.413} C_VEL
LIN {X 0,Y 254.011,Z 281.163,A -85,B 0,C 180,E1 -19923.063,E2 -19923.063} C_VEL
LIN {X 0,Y 256.173,Z 242.337,A -85,B 0,C 180,E1 -19924.262,E2 -19924.262} C_VEL
LIN {X 0,Y 254.987,Z 234.787,A -85,B 0,C 180,E1 -19924.825,E2 -19924.825} C_VEL
LIN {X 0,Y 250.06,Z 223.26,A -85,B 0,C 180,E1 -19926.392,E2 -19926.392} C_VEL
LIN {X 0,Y 244.793,Z 212.728,A -85,B 0,C 180,E1 -19928.132,E2 -19928.132} C_VEL
LIN {X 0,Y 239.704,Z 203.835,A -85,B 0,C 180,E1 -19929.903,E2 -19929.903} C_VEL
LIN {X 0,Y 236.435,Z 198.664,A -85,B 0,C 180,E1 -19931.11,E2 -19931.11} C_VEL
LIN {X 0,Y 233.286,Z 193.783,A -85,B 0,C 180,E1 -19932.348,E2 -19932.348} C_VEL
LIN {X 0,Y 230.209,Z 189.091,A -85,B 0,C 180,E1 -19933.684,E2 -19933.684} C_VEL
LIN {X 0,Y 229.403,Z 186.629,A -85,B 0,C 180,E1 -19935.199,E2 -19935.199} C_VEL
LIN {X 0,Y 227.812,Z 181.66,A -85,B 0,C 180,E1 -19939.229,E2 -19939.229} C_VEL
LIN {X 0,Y 227.873,Z 181.601,A -85,B 0,C 180,E1 -19944.126,E2 -19944.126} C_VEL
LIN {X 0,Y 227.848,Z 181.595,A -85,B 0,C 180,E1 -19948.373,E2 -19948.373} C_VEL
LIN {X 0,Y 227.846,Z 181.593,A -85,B 0,C 180,E1 -19952.439,E2 -19952.439} C_VEL
LIN {X 0,Y 227.881,Z 181.587,A -85,B 0,C 180,E1 -19956.363,E2 -19956.363} C_VEL
LIN {X 0,Y 227.883,Z 181.587,A -85,B 0,C 180,E1 -19960.168,E2 -19960.168} C_VEL
LIN {X 0,Y 228.008,Z 181.573,A -85,B 0,C 180,E1 -19963.893,E2 -19963.893} C_VEL
LIN {X 0,Y 228.117,Z 181.559,A -85,B 0,C 180,E1 -19969.347,E2 -19969.347} C_VEL
LIN {X 0,Y 228.298,Z 181.536,A -85,B 0,C 180,E1 -19972.926,E2 -19972.926} C_VEL
LIN {X 0,Y 228.525,Z 181.519,A -85,B 0,C 180,E1 -19978.237,E2 -19978.237} C_VEL
LIN {X 0,Y 228.526,Z 181.52,A -85,B 0,C 180,E1 -19981.762,E2 -19981.762} C_VEL
LIN {X 0,Y 228.299,Z 181.701,A -85,B 0,C 180,E1 -19987.517,E2 -19987.517} C_VEL
LIN {X 0,Y 229.25,Z 184.952,A -85,B 0,C 180,E1 -19989.975,E2 -19989.975} C_VEL
LIN {X 0,Y 232.078,Z 189.376,A -85,B 0,C 180,E1 -19991.296,E2 -19991.296} C_VEL
LIN {X 0,Y 237.146,Z 196.664,A -85,B 0,C 180,E1 -19993.274,E2 -19993.274} C_VEL
LIN {X 0,Y 240.71,Z 202.458,A -85,B 0,C 180,E1 -19994.585,E2 -19994.585} C_VEL
LIN {X 0,Y 246.226,Z 211.876,A -85,B 0,C 180,E1 -19996.464,E2 -19996.464} C_VEL
LIN {X 0,Y 252.005,Z 223.311,A -85,B 0,C 180,E1 -19998.321,E2 -19998.321} C_VEL
LIN {X 0,Y 256.629,Z 234.277,A -85,B 0,C 180,E1 -19999.77,E2 -19999.77} C_VEL
LIN {X 0,Y 253.094,Z 293.019,A -85,B 0,C 180,E1 -20001.602,E2 -20001.602} C_VEL
LIN {X 0,Y 251.483,Z 306.748,A -85,B 0,C 180,E1 -20002.329,E2 -20002.329} C_VEL
LIN {X 0,Y 249.455,Z 319.694,A -85,B 0,C 180,E1 -20003.375,E2 -20003.375} C_VEL
LIN {X 0,Y 246.974,Z 331.602,A -85,B 0,C 180,E1 -20004.666,E2 -20004.666} C_VEL
LIN {X 0,Y 244.377,Z 342.131,A -85,B 0,C 180,E1 -20006.141,E2 -20006.141} C_VEL
LIN {X 0,Y 241.537,Z 352.039,A -85,B 0,C 180,E1 -20007.886,E2 -20007.886} C_VEL
LIN {X 0,Y 238.323,Z 361.884,A -85,B 0,C 180,E1 -20010.086,E2 -20010.086} C_VEL
LIN {X 0,Y 235.397,Z 370.382,A -85,B 0,C 180,E1 -20012.506,E2 -20012.506} C_VEL
LIN {X 0,Y 232.451,Z 378.009,A -85,B 0,C 180,E1 -20015.286,E2 -20015.286} C_VEL
LIN {X 0,Y 230.139,Z 384.021,A -85,B 0,C 180,E1 -20018.158,E2 -20018.158} C_VEL
LIN {X 0,Y 228.2,Z 388.775,A -85,B 0,C 180,E1 -20021.187,E2 -20021.187} C_VEL
LIN {X 0,Y 226.748,Z 392.336,A -85,B 0,C 180,E1 -20024.534,E2 -20024.534} C_VEL
LIN {X 0,Y 226.075,Z 393.942,A -85,B 0,C 180,E1 -20026.853,E2 -20026.853} C_VEL
LIN {X 0,Y 225.568,Z 394.806,A -85,B 0,C 180,E1 -20029.137,E2 -20029.137} C_VEL
LIN {X 0,Y 225.236,Z 395.061,A -85,B 0,C 180,E1 -20031.39,E2 -20031.39} C_VEL
LIN {X 0,Y 225.093,Z 394.437,A -85,B 0,C 180,E1 -20034.269,E2 -20034.269} C_VEL
LIN {X 0,Y 225.277,Z 392.561,A -85,B 0,C 180,E1 -20037.385,E2 -20037.385} C_VEL
LIN {X 0,Y 225.836,Z 389.25,A -85,B 0,C 180,E1 -20040.615,E2 -20040.615} C_VEL
LIN {X 0,Y 226.403,Z 385.486,A -85,B 0,C 180,E1 -20043.206,E2 -20043.206} C_VEL
LIN {X 0,Y 227.37,Z 379.536,A -85,B 0,C 180,E1 -20046.31,E2 -20046.31} C_VEL
LIN {X 0,Y 228.563,Z 373.302,A -85,B 0,C 180,E1 -20048.823,E2 -20048.823} C_VEL
LIN {X 0,Y 230.02,Z 365.685,A -85,B 0,C 180,E1 -20051.29,E2 -20051.29} C_VEL
LIN {X 0,Y 231.915,Z 356.294,A -85,B 0,C 180,E1 -20053.723,E2 -20053.723} C_VEL
LIN {X 0,Y 233.738,Z 346.692,A -85,B 0,C 180,E1 -20055.715,E2 -20055.715} C_VEL
LIN {X 0,Y 235.669,Z 335.731,A -85,B 0,C 180,E1 -20057.516,E2 -20057.516} C_VEL
LIN {X 0,Y 237.286,Z 324.54,A -85,B 0,C 180,E1 -20058.974,E2 -20058.974} C_VEL
LIN {X 0,Y 238.719,Z 312.829,A -85,B 0,C 180,E1 -20060.149,E2 -20060.149} C_VEL
LIN {X 0,Y 240.002,Z 299.779,A -85,B 0,C 180,E1 -20061.079,E2 -20061.079} C_VEL
LIN {X 0,Y 240.886,Z 286.525,A -85,B 0,C 180,E1 -20061.684,E2 -20061.684} C_VEL
LIN {X 0,Y 243.207,Z 224.866,A -85,B 0,C 180,E1 -20063.638,E2 -20063.638} C_VEL
LIN {X 0,Y 242.115,Z 219.139,A -85,B 0,C 180,E1 -20063.959,E2 -20063.959} C_VEL
LIN {X 0,Y 234.424,Z 197.867,A -85,B 0,C 180,E1 -20065.594,E2 -20065.594} C_VEL
LIN {X 0,Y 228.91,Z 184.376,A -85,B 0,C 180,E1 -20066.812,E2 -20066.812} C_VEL
LIN {X 0,Y 228.697,Z 183.236,A -85,B 0,C 180,E1 -20067.14,E2 -20067.14} C_VEL
LIN {X 0,Y 228.504,Z 181.548,A -85,B 0,C 180,E1 -20068.019,E2 -20068.019} C_VEL
LIN {X 0,Y 228.618,Z 181.504,A -85,B 0,C 180,E1 -20070.002,E2 -20070.002} C_VEL
LIN {X 0,Y 228.552,Z 181.513,A -85,B 0,C 180,E1 -20071.764,E2 -20071.764} C_VEL
LIN {X 0,Y 228.317,Z 181.541,A -85,B 0,C 180,E1 -20077.074,E2 -20077.074} C_VEL
LIN {X 0,Y 228.142,Z 181.566,A -85,B 0,C 180,E1 -20080.653,E2 -20080.653} C_VEL
LIN {X 0,Y 228.057,Z 181.575,A -85,B 0,C 180,E1 -20084.274,E2 -20084.274} C_VEL
LIN {X 0,Y 228.003,Z 181.574,A -85,B 0,C 180,E1 -20087.955,E2 -20087.955} C_VEL
LIN {X 0,Y 227.93,Z 181.592,A -85,B 0,C 180,E1 -20092.331,E2 -20092.331} C_VEL
LIN {X 0,Y 227.942,Z 181.573,A -85,B 0,C 180,E1 -20096.604,E2 -20096.604} C_VEL
LIN {X 0,Y 227.897,Z 181.596,A -85,B 0,C 180,E1 -20100.292,E2 -20100.292} C_VEL
LIN {X 0,Y 227.877,Z 181.59,A -85,B 0,C 180,E1 -20103.722,E2 -20103.722} C_VEL
LIN {X 0,Y 227.844,Z 181.589,A -85,B 0,C 180,E1 -20108.093,E2 -20108.093} C_VEL
LIN {X 0,Y 227.814,Z 181.608,A -85,B 0,C 180,E1 -20112.743,E2 -20112.743} C_VEL
LIN {X 0,Y 227.814,Z 181.58,A -85,B 0,C 180,E1 -20117.259,E2 -20117.259} C_VEL
LIN {X 0,Y 227.841,Z 181.593,A -85,B 0,C 180,E1 -20121.909,E2 -20121.909} C_VEL
LIN {X 0,Y 227.88,Z 181.6,A -85,B 0,C 180,E1 -20126.379,E2 -20126.379} C_VEL
LIN {X 0,Y 227.878,Z 181.594,A -85,B 0,C 180,E1 -20130.433,E2 -20130.433} C_VEL
LIN {X 0,Y 227.905,Z 181.594,A -85,B 0,C 180,E1 -20134.424,E2 -20134.424} C_VEL
LIN {X 0,Y 227.958,Z 181.583,A -85,B 0,C 180,E1 -20138.288,E2 -20138.288} C_VEL
LIN {X 0,Y 228.038,Z 181.574,A -85,B 0,C 180,E1 -20142.828,E2 -20142.828} C_VEL
LIN {X 0,Y 228.074,Z 181.572,A -85,B 0,C 180,E1 -20147.544,E2 -20147.544} C_VEL
LIN {X 0,Y 228.256,Z 181.546,A -85,B 0,C 180,E1 -20151.145,E2 -20151.145} C_VEL
LIN {X 0,Y 228.303,Z 181.538,A -85,B 0,C 180,E1 -20152.928,E2 -20152.928} C_VEL
LIN {X 0,Y 228.539,Z 181.512,A -85,B 0,C 180,E1 -20158.239,E2 -20158.239} C_VEL
LIN {X 0,Y 228.538,Z 181.49,A -85,B 0,C 180,E1 -20161.763,E2 -20161.763} C_VEL
LIN {X 0,Y 228.309,Z 181.536,A -85,B 0,C 180,E1 -20167.074,E2 -20167.074} C_VEL
LIN {X 0,Y 228.147,Z 181.564,A -85,B 0,C 180,E1 -20170.652,E2 -20170.652} C_VEL
LIN {X 0,Y 228.036,Z 181.563,A -85,B 0,C 180,E1 -20174.275,E2 -20174.275} C_VEL
LIN {X 0,Y 227.93,Z 181.58,A -85,B 0,C 180,E1 -20177.96,E2 -20177.96} C_VEL
LIN {X 0,Y 227.893,Z 181.596,A -85,B 0,C 180,E1 -20182.303,E2 -20182.303} C_VEL
LIN {X 0,Y 227.893,Z 181.58,A -85,B 0,C 180,E1 -20186.742,E2 -20186.742} C_VEL
LIN {X 0,Y 227.877,Z 181.599,A -85,B 0,C 180,E1 -20190.28,E2 -20190.28} C_VEL
LIN {X 0,Y 227.842,Z 181.589,A -85,B 0,C 180,E1 -20194.428,E2 -20194.428} C_VEL
LIN {X 0,Y 227.149,Z 181.688,A -85,B 0,C 180,E1 -20195.904,E2 -20195.904} C_VEL
LIN {X 0,Y 224.289,Z 182.046,A -85,B 0,C 180,E1 -20198.313,E2 -20198.313} C_VEL
LIN {X 0,Y 221.87,Z 182.347,A -85,B 0,C 180,E1 -20200.279,E2 -20200.279} C_VEL
LIN {X 0,Y 220.831,Z 182.476,A -85,B 0,C 180,E1 -20201.805,E2 -20201.805} C_VEL
LIN {X 0,Y 220.744,Z 182.487,A -85,B 0,C 180,E1 -20202.322,E2 -20202.322} C_VEL
LIN {X 0,Y 220.757,Z 182.479,A -85,B 0,C 180,E1 -20205.54,E2 -20205.54} C_VEL
LIN {X 0,Y 220.785,Z 182.482,A -85,B 0,C 180,E1 -20210.457,E2 -20210.457} C_VEL
LIN {X 0,Y 220.836,Z 182.705,A -85,B 0,C 180,E1 -20212.882,E2 -20212.882} C_VEL
LIN {X 0,Y 222.593,Z 190.359,A -85,B 0,C 180,E1 -20216.389,E2 -20216.389} C_VEL
LIN {X 0,Y 230.3,Z 210.048,A -85,B 0,C 180,E1 -20218.167,E2 -20218.167} C_VEL
LIN {X 0,Y 233.821,Z 220.433,A -85,B 0,C 180,E1 -20218.963,E2 -20218.963} C_VEL
LIN {X 0,Y 236.402,Z 239.943,A -85,B 0,C 180,E1 -20219.968,E2 -20219.968} C_VEL
LIN {X 0,Y 233.885,Z 299.32,A -85,B 0,C 180,E1 -20221.935,E2 -20221.935} C_VEL
LIN {X 0,Y 232.702,Z 312.525,A -85,B 0,C 180,E1 -20222.696,E2 -20222.696} C_VEL
LIN {X 0,Y 231.31,Z 324.775,A -85,B 0,C 180,E1 -20223.737,E2 -20223.737} C_VEL
LIN {X 0,Y 229.544,Z 336.618,A -85,B 0,C 180,E1 -20225.102,E2 -20225.102} C_VEL
LIN {X 0,Y 227.779,Z 346.759,A -85,B 0,C 180,E1 -20226.592,E2 -20226.592} C_VEL
LIN {X 0,Y 225.796,Z 357.568,A -85,B 0,C 180,E1 -20228.594,E2 -20228.594} C_VEL
LIN {X 0,Y 223.999,Z 366.963,A -85,B 0,C 180,E1 -20230.785,E2 -20230.785} C_VEL
LIN {X 0,Y 222.142,Z 376.067,A -85,B 0,C 180,E1 -20233.455,E2 -20233.455} C_VEL
LIN {X 0,Y 220.579,Z 383.437,A -85,B 0,C 180,E1 -20236.173,E2 -20236.173} C_VEL
LIN {X 0,Y 219.591,Z 389.322,A -85,B 0,C 180,E1 -20238.927,E2 -20238.927} C_VEL
LIN {X 0,Y 218.904,Z 393.918,A -85,B 0,C 180,E1 -20241.691,E2 -20241.691} C_VEL
LIN {X 0,Y 218.571,Z 397.39,A -85,B 0,C 180,E1 -20244.463,E2 -20244.463} C_VEL
LIN {X 0,Y 218.501,Z 399.104,A -85,B 0,C 180,E1 -20246.31,E2 -20246.31} C_VEL
LIN {X 0,Y 218.475,Z 400.401,A -85,B 0,C 180,E1 -20248.155,E2 -20248.155} C_VEL
LIN {X 0,Y 218.576,Z 401.295,A -85,B 0,C 180,E1 -20249.998,E2 -20249.998} C_VEL
LIN {X 0,Y 218.474,Z 401.753,A -85,B 0,C 180,E1 -20251.841,E2 -20251.841} C_VEL
LIN {X 0,Y 218.515,Z 401.722,A -85,B 0,C 180,E1 -20254.401,E2 -20254.401} C_VEL
LIN {X 0,Y 218.859,Z 400.721,A -85,B 0,C 180,E1 -20257.378,E2 -20257.378} C_VEL
LIN {X 0,Y 219.238,Z 399.582,A -85,B 0,C 180,E1 -20259.221,E2 -20259.221} C_VEL
LIN {X 0,Y 219.837,Z 398.004,A -85,B 0,C 180,E1 -20261.057,E2 -20261.057} C_VEL
LIN {X 0,Y 221.036,Z 394.859,A -85,B 0,C 180,E1 -20263.794,E2 -20263.794} C_VEL
LIN {X 0,Y 222.66,Z 390.685,A -85,B 0,C 180,E1 -20266.501,E2 -20266.501} C_VEL
LIN {X 0,Y 225.447,Z 384.343,A -85,B 0,C 180,E1 -20269.577,E2 -20269.577} C_VEL
LIN {X 0,Y 227.935,Z 377.434,A -85,B 0,C 180,E1 -20272.214,E2 -20272.214} C_VEL
LIN {X 0,Y 231.104,Z 368.963,A -85,B 0,C 180,E1 -20274.715,E2 -20274.715} C_VEL
LIN {X 0,Y 234.085,Z 360.251,A -85,B 0,C 180,E1 -20276.764,E2 -20276.764} C_VEL
LIN {X 0,Y 237.471,Z 349.573,A -85,B 0,C 180,E1 -20278.743,E2 -20278.743} C_VEL
LIN {X 0,Y 240.339,Z 338.984,A -85,B 0,C 180,E1 -20280.291,E2 -20280.291} C_VEL
LIN {X 0,Y 243.069,Z 327.278,A -85,B 0,C 180,E1 -20281.602,E2 -20281.602} C_VEL
LIN {X 0,Y 245.506,Z 314.077,A -85,B 0,C 180,E1 -20282.703,E2 -20282.703} C_VEL
LIN {X 0,Y 247.234,Z 300.687,A -85,B 0,C 180,E1 -20283.465,E2 -20283.465} C_VEL
LIN {X 0,Y 248.673,Z 281.007,A -85,B 0,C 180,E1 -20284.134,E2 -20284.134} C_VEL
LIN {X 0,Y 250.873,Z 243.466,A -85,B 0,C 180,E1 -20285.313,E2 -20285.313} C_VEL
LIN {X 0,Y 249.942,Z 237.778,A -85,B 0,C 180,E1 -20285.766,E2 -20285.766} C_VEL
LIN {X 0,Y 245.228,Z 226.654,A -85,B 0,C 180,E1 -20287.355,E2 -20287.355} C_VEL
LIN {X 0,Y 240.479,Z 217.002,A -85,B 0,C 180,E1 -20289.029,E2 -20289.029} C_VEL
LIN {X 0,Y 235.903,Z 208.848,A -85,B 0,C 180,E1 -20290.716,E2 -20290.716} C_VEL
LIN {X 0,Y 232.725,Z 203.682,A -85,B 0,C 180,E1 -20291.963,E2 -20291.963} C_VEL
LIN {X 0,Y 229.662,Z 198.94,A -85,B 0,C 180,E1 -20293.222,E2 -20293.222} C_VEL
LIN {X 0,Y 226.204,Z 193.774,A -85,B 0,C 180,E1 -20294.761,E2 -20294.761} C_VEL
LIN {X 0,Y 222.729,Z 188.572,A -85,B 0,C 180,E1 -20296.547,E2 -20296.547} C_VEL
LIN {X 0,Y 221.081,Z 183.759,A -85,B 0,C 180,E1 -20300.521,E2 -20300.521} C_VEL
LIN {X 0,Y 220.801,Z 182.501,A -85,B 0,C 180,E1 -20301.925,E2 -20301.925} C_VEL
LIN {X 0,Y 220.8,Z 182.472,A -85,B 0,C 180,E1 -20305.845,E2 -20305.845} C_VEL
LIN {X 0,Y 220.827,Z 182.467,A -85,B 0,C 180,E1 -20309.388,E2 -20309.388} C_VEL
LIN {X 0,Y 220.867,Z 182.463,A -85,B 0,C 180,E1 -20313.545,E2 -20313.545} C_VEL
LIN {X 0,Y 220.845,Z 182.465,A -85,B 0,C 180,E1 -20317.549,E2 -20317.549} C_VEL
LIN {X 0,Y 220.911,Z 182.466,A -85,B 0,C 180,E1 -20322.624,E2 -20322.624} C_VEL
LIN {X 0,Y 220.976,Z 182.459,A -85,B 0,C 180,E1 -20327.136,E2 -20327.136} C_VEL
LIN {X 0,Y 221.186,Z 182.435,A -85,B 0,C 180,E1 -20330.858,E2 -20330.858} C_VEL
LIN {X 0,Y 221.235,Z 182.415,A -85,B 0,C 180,E1 -20332.699,E2 -20332.699} C_VEL
LIN {X 0,Y 221.459,Z 182.399,A -85,B 0,C 180,E1 -20338.181,E2 -20338.181} C_VEL
LIN {X 0,Y 221.459,Z 182.401,A -85,B 0,C 180,E1 -20341.818,E2 -20341.818} C_VEL
LIN {X 0,Y 221.149,Z 182.662,A -85,B 0,C 180,E1 -20345.013,E2 -20345.013} C_VEL
LIN {X 0,Y 222.259,Z 185.374,A -85,B 0,C 180,E1 -20347.38,E2 -20347.38} C_VEL
LIN {X 0,Y 225.029,Z 189.546,A -85,B 0,C 180,E1 -20348.813,E2 -20348.813} C_VEL
LIN {X 0,Y 226.768,Z 191.892,A -85,B 0,C 180,E1 -20349.611,E2 -20349.611} C_VEL
LIN {X 0,Y 230.476,Z 197.324,A -85,B 0,C 180,E1 -20351.236,E2 -20351.236} C_VEL
LIN {X 0,Y 234.282,Z 203.082,A -85,B 0,C 180,E1 -20352.766,E2 -20352.766} C_VEL
LIN {X 0,Y 238.807,Z 210.582,A -85,B 0,C 180,E1 -20354.483,E2 -20354.483} C_VEL
LIN {X 0,Y 244.733,Z 221.679,A -85,B 0,C 180,E1 -20356.567,E2 -20356.567} C_VEL
LIN {X 0,Y 248.854,Z 230.597,A -85,B 0,C 180,E1 -20357.953,E2 -20357.953} C_VEL
LIN {X 0,Y 251.254,Z 236.4,A -85,B 0,C 180,E1 -20358.739,E2 -20358.739} C_VEL
LIN {X 0,Y 247.784,Z 292.409,A -85,B 0,C 180,E1 -20360.516,E2 -20360.516} C_VEL
LIN {X 0,Y 246.07,Z 306.382,A -85,B 0,C 180,E1 -20361.25,E2 -20361.25} C_VEL
LIN {X 0,Y 243.936,Z 319.546,A -85,B 0,C 180,E1 -20362.322,E2 -20362.322} C_VEL
LIN {X 0,Y 241.292,Z 331.654,A -85,B 0,C 180,E1 -20363.653,E2 -20363.653} C_VEL
LIN {X 0,Y 238.217,Z 343.475,A -85,B 0,C 180,E1 -20365.362,E2 -20365.362} C_VEL
LIN {X 0,Y 235.126,Z 353.54,A -85,B 0,C 180,E1 -20367.228,E2 -20367.228} C_VEL
LIN {X 0,Y 231.859,Z 362.974,A -85,B 0,C 180,E1 -20369.431,E2 -20369.431} C_VEL
LIN {X 0,Y 228.818,Z 371.218,A -85,B 0,C 180,E1 -20371.882,E2 -20371.882} C_VEL
LIN {X 0,Y 225.684,Z 378.815,A -85,B 0,C 180,E1 -20374.796,E2 -20374.796} C_VEL
LIN {X 0,Y 223.62,Z 383.855,A -85,B 0,C 180,E1 -20377.294,E2 -20377.294} C_VEL
LIN {X 0,Y 221.502,Z 388.664,A -85,B 0,C 180,E1 -20380.408,E2 -20380.408} C_VEL
LIN {X 0,Y 220.296,Z 391.364,A -85,B 0,C 180,E1 -20382.801,E2 -20382.801} C_VEL
LIN {X 0,Y 219.426,Z 393.335,A -85,B 0,C 180,E1 -20385.203,E2 -20385.203} C_VEL
LIN {X 0,Y 218.789,Z 394.583,A -85,B 0,C 180,E1 -20387.629,E2 -20387.629} C_VEL
LIN {X 0,Y 218.237,Z 395.172,A -85,B 0,C 180,E1 -20390.612,E2 -20390.612} C_VEL
LIN {X 0,Y 218.006,Z 394.686,A -85,B 0,C 180,E1 -20393.7,E2 -20393.7} C_VEL
LIN {X 0,Y 218.128,Z 392.986,A -85,B 0,C 180,E1 -20396.897,E2 -20396.897} C_VEL
LIN {X 0,Y 218.651,Z 389.855,A -85,B 0,C 180,E1 -20400.208,E2 -20400.208} C_VEL
LIN {X 0,Y 219.341,Z 385.521,A -85,B 0,C 180,E1 -20403.35,E2 -20403.35} C_VEL
LIN {X 0,Y 220.331,Z 379.645,A -85,B 0,C 180,E1 -20406.505,E2 -20406.505} C_VEL
LIN {X 0,Y 221.568,Z 373.413,A -85,B 0,C 180,E1 -20409.096,E2 -20409.096} C_VEL
LIN {X 0,Y 223.057,Z 365.805,A -85,B 0,C 180,E1 -20411.637,E2 -20411.637} C_VEL
LIN {X 0,Y 224.897,Z 357.035,A -85,B 0,C 180,E1 -20413.991,E2 -20413.991} C_VEL
LIN {X 0,Y 226.832,Z 347.247,A -85,B 0,C 180,E1 -20416.109,E2 -20416.109} C_VEL
LIN {X 0,Y 228.684,Z 337.173,A -85,B 0,C 180,E1 -20417.846,E2 -20417.846} C_VEL
LIN {X 0,Y 230.495,Z 325.326,A -85,B 0,C 180,E1 -20419.461,E2 -20419.461} C_VEL
LIN {X 0,Y 232.078,Z 312.966,A -85,B 0,C 180,E1 -20420.744,E2 -20420.744} C_VEL
LIN {X 0,Y 233.363,Z 300.239,A -85,B 0,C 180,E1 -20421.682,E2 -20421.682} C_VEL
LIN {X 0,Y 234.314,Z 286.531,A -85,B 0,C 180,E1 -20422.328,E2 -20422.328} C_VEL
LIN {X 0,Y 236.705,Z 225.86,A -85,B 0,C 180,E1 -20424.301,E2 -20424.301} C_VEL
LIN {X 0,Y 235.862,Z 221.502,A -85,B 0,C 180,E1 -20424.554,E2 -20424.554} C_VEL
LIN {X 0,Y 228.456,Z 200.809,A -85,B 0,C 180,E1 -20426.191,E2 -20426.191} C_VEL
LIN {X 0,Y 221.804,Z 184.354,A -85,B 0,C 180,E1 -20427.726,E2 -20427.726} C_VEL
LIN {X 0,Y 221.548,Z 182.516,A -85,B 0,C 180,E1 -20428.468,E2 -20428.468} C_VEL
LIN {X 0,Y 221.509,Z 182.391,A -85,B 0,C 180,E1 -20431.82,E2 -20431.82} C_VEL
LIN {X 0,Y 221.252,Z 182.419,A -85,B 0,C 180,E1 -20437.301,E2 -20437.301} C_VEL
LIN {X 0,Y 221.063,Z 182.449,A -85,B 0,C 180,E1 -20440.998,E2 -20440.998} C_VEL
LIN {X 0,Y 221.016,Z 182.454,A -85,B 0,C 180,E1 -20446.632,E2 -20446.632} C_VEL
LIN {X 0,Y 220.893,Z 182.463,A -85,B 0,C 180,E1 -20450.488,E2 -20450.488} C_VEL
LIN {X 0,Y 220.868,Z 182.467,A -85,B 0,C 180,E1 -20454.437,E2 -20454.437} C_VEL
LIN {X 0,Y 220.827,Z 182.469,A -85,B 0,C 180,E1 -20458.517,E2 -20458.517} C_VEL
LIN {X 0,Y 220.817,Z 182.476,A -85,B 0,C 180,E1 -20462.758,E2 -20462.758} C_VEL
LIN {X 0,Y 220.81,Z 182.457,A -85,B 0,C 180,E1 -20467.279,E2 -20467.279} C_VEL
LIN {X 0,Y 220.772,Z 182.483,A -85,B 0,C 180,E1 -20471.954,E2 -20471.954} C_VEL
LIN {X 0,Y 220.777,Z 182.47,A -85,B 0,C 180,E1 -20475.548,E2 -20475.548} C_VEL
LIN {X 0,Y 220.808,Z 182.457,A -85,B 0,C 180,E1 -20480.465,E2 -20480.465} C_VEL
LIN {X 0,Y 220.827,Z 182.471,A -85,B 0,C 180,E1 -20482.794,E2 -20482.794} C_VEL
LIN {X 0,Y 220.814,Z 182.475,A -85,B 0,C 180,E1 -20487.244,E2 -20487.244} C_VEL
LIN {X 0,Y 220.806,Z 182.477,A -85,B 0,C 180,E1 -20491.483,E2 -20491.483} C_VEL
LIN {X 0,Y 220.85,Z 182.47,A -85,B 0,C 180,E1 -20495.564,E2 -20495.564} C_VEL
LIN {X 0,Y 220.89,Z 182.466,A -85,B 0,C 180,E1 -20499.515,E2 -20499.515} C_VEL
LIN {X 0,Y 221.018,Z 182.447,A -85,B 0,C 180,E1 -20503.371,E2 -20503.371} C_VEL
LIN {X 0,Y 221.071,Z 182.445,A -85,B 0,C 180,E1 -20509.005,E2 -20509.005} C_VEL
LIN {X 0,Y 221.241,Z 182.417,A -85,B 0,C 180,E1 -20512.701,E2 -20512.701} C_VEL
LIN {X 0,Y 221.472,Z 182.393,A -85,B 0,C 180,E1 -20518.182,E2 -20518.182} C_VEL
LIN {X 0,Y 221.472,Z 182.368,A -85,B 0,C 180,E1 -20521.819,E2 -20521.819} C_VEL
LIN {X 0,Y 221.247,Z 182.417,A -85,B 0,C 180,E1 -20527.301,E2 -20527.301} C_VEL
LIN {X 0,Y 221.067,Z 182.447,A -85,B 0,C 180,E1 -20530.997,E2 -20530.997} C_VEL
LIN {X 0,Y 220.98,Z 182.433,A -85,B 0,C 180,E1 -20536.633,E2 -20536.633} C_VEL
LIN {X 0,Y 220.852,Z 182.473,A -85,B 0,C 180,E1 -20540.491,E2 -20540.491} C_VEL
LIN {X 0,Y 220.801,Z 182.469,A -85,B 0,C 180,E1 -20544.444,E2 -20544.444} C_VEL
LIN {X 0,Y 220.803,Z 182.476,A -85,B 0,C 180,E1 -20548.519,E2 -20548.519} C_VEL
LIN {X 0,Y 220.817,Z 182.468,A -85,B 0,C 180,E1 -20552.757,E2 -20552.757} C_VEL
LIN {X 0,Y 220.807,Z 182.481,A -85,B 0,C 180,E1 -20557.275,E2 -20557.275} C_VEL
LIN {X 0,Y 220.753,Z 182.486,A -85,B 0,C 180,E1 -20561.958,E2 -20561.958} C_VEL
LIN {X 0,Y 220.744,Z 182.487,A -85,B 0,C 180,E1 -20562.322,E2 -20562.322} C_VEL
LIN {X 0,Y 220.062,Z 182.573,A -85,B 0,C 180,E1 -20563.843,E2 -20563.843} C_VEL
LIN {X 0,Y 217.187,Z 182.929,A -85,B 0,C 180,E1 -20566.325,E2 -20566.325} C_VEL
LIN {X 0,Y 214.766,Z 183.23,A -85,B 0,C 180,E1 -20568.352,E2 -20568.352} C_VEL
LIN {X 0,Y 213.755,Z 183.36,A -85,B 0,C 180,E1 -20569.927,E2 -20569.927} C_VEL
LIN {X 0,Y 213.687,Z 183.36,A -85,B 0,C 180,E1 -20570.461,E2 -20570.461} C_VEL
LIN {X 0,Y 213.772,Z 183.433,A -85,B 0,C 180,E1 -20572.096,E2 -20572.096} C_VEL
LIN {X 0,Y 215.296,Z 190.01,A -85,B 0,C 180,E1 -20575.338,E2 -20575.338} C_VEL
LIN {X 0,Y 216.414,Z 193.068,A -85,B 0,C 180,E1 -20575.741,E2 -20575.741} C_VEL
LIN {X 0,Y 224.453,Z 213.396,A -85,B 0,C 180,E1 -20577.596,E2 -20577.596} C_VEL
LIN {X 0,Y 227.621,Z 223.039,A -85,B 0,C 180,E1 -20578.354,E2 -20578.354} C_VEL
LIN {X 0,Y 229.878,Z 240.563,A -85,B 0,C 180,E1 -20579.285,E2 -20579.285} C_VEL
LIN {X 0,Y 227.373,Z 298.423,A -85,B 0,C 180,E1 -20581.246,E2 -20581.246} C_VEL
LIN {X 0,Y 226.129,Z 311.856,A -85,B 0,C 180,E1 -20582.022,E2 -20582.022} C_VEL
LIN {X 0,Y 224.62,Z 324.791,A -85,B 0,C 180,E1 -20583.144,E2 -20583.144} C_VEL
LIN {X 0,Y 222.812,Z 336.607,A -85,B 0,C 180,E1 -20584.546,E2 -20584.546} C_VEL
LIN {X 0,Y 220.989,Z 346.731,A -85,B 0,C 180,E1 -20586.077,E2 -20586.077} C_VEL
LIN {X 0,Y 218.985,Z 357.312,A -85,B 0,C 180,E1 -20588.092,E2 -20588.092} C_VEL
LIN {X 0,Y 217.146,Z 366.54,A -85,B 0,C 180,E1 -20590.291,E2 -20590.291} C_VEL
LIN {X 0,Y 215.272,Z 375.313,A -85,B 0,C 180,E1 -20592.911,E2 -20592.911} C_VEL
LIN {X 0,Y 213.656,Z 382.8,A -85,B 0,C 180,E1 -20595.716,E2 -20595.716} C_VEL
LIN {X 0,Y 212.577,Z 388.797,A -85,B 0,C 180,E1 -20598.557,E2 -20598.557} C_VEL
LIN {X 0,Y 211.864,Z 393.498,A -85,B 0,C 180,E1 -20601.413,E2 -20601.413} C_VEL
LIN {X 0,Y 211.494,Z 397.049,A -85,B 0,C 180,E1 -20604.277,E2 -20604.277} C_VEL
LIN {X 0,Y 211.4,Z 398.824,A -85,B 0,C 180,E1 -20606.186,E2 -20606.186} C_VEL
LIN {X 0,Y 211.382,Z 400.159,A -85,B 0,C 180,E1 -20608.093,E2 -20608.093} C_VEL
LIN {X 0,Y 211.475,Z 401.091,A -85,B 0,C 180,E1 -20609.998,E2 -20609.998} C_VEL
LIN {X 0,Y 211.38,Z 401.615,A -85,B 0,C 180,E1 -20611.903,E2 -20611.903} C_VEL
LIN {X 0,Y 211.421,Z 401.658,A -85,B 0,C 180,E1 -20614.239,E2 -20614.239} C_VEL
LIN {X 0,Y 211.819,Z 400.699,A -85,B 0,C 180,E1 -20617.625,E2 -20617.625} C_VEL
LIN {X 0,Y 212.223,Z 399.621,A -85,B 0,C 180,E1 -20619.529,E2 -20619.529} C_VEL
LIN {X 0,Y 212.846,Z 398.104,A -85,B 0,C 180,E1 -20621.425,E2 -20621.425} C_VEL
LIN {X 0,Y 214.139,Z 395.055,A -85,B 0,C 180,E1 -20624.247,E2 -20624.247} C_VEL
LIN {X 0,Y 215.875,Z 390.975,A -85,B 0,C 180,E1 -20627.036,E2 -20627.036} C_VEL
LIN {X 0,Y 218.798,Z 384.729,A -85,B 0,C 180,E1 -20630.198,E2 -20630.198} C_VEL
LIN {X 0,Y 221.359,Z 378.029,A -85,B 0,C 180,E1 -20632.87,E2 -20632.87} C_VEL
LIN {X 0,Y 224.719,Z 369.642,A -85,B 0,C 180,E1 -20635.467,E2 -20635.467} C_VEL
LIN {X 0,Y 227.822,Z 361.129,A -85,B 0,C 180,E1 -20637.561,E2 -20637.561} C_VEL
LIN {X 0,Y 231.332,Z 350.693,A -85,B 0,C 180,E1 -20639.58,E2 -20639.58} C_VEL
LIN {X 0,Y 234.715,Z 339.014,A -85,B 0,C 180,E1 -20641.347,E2 -20641.347} C_VEL
LIN {X 0,Y 237.56,Z 327.345,A -85,B 0,C 180,E1 -20642.675,E2 -20642.675} C_VEL
LIN {X 0,Y 240.089,Z 314.2,A -85,B 0,C 180,E1 -20643.789,E2 -20643.789} C_VEL
LIN {X 0,Y 241.917,Z 300.819,A -85,B 0,C 180,E1 -20644.562,E2 -20644.562} C_VEL
LIN {X 0,Y 243.379,Z 281.878,A -85,B 0,C 180,E1 -20645.219,E2 -20645.219} C_VEL
LIN {X 0,Y 245.646,Z 244.44,A -85,B 0,C 180,E1 -20646.421,E2 -20646.421} C_VEL
LIN {X 0,Y 245.054,Z 240.973,A -85,B 0,C 180,E1 -20646.719,E2 -20646.719} C_VEL
LIN {X 0,Y 240.171,Z 229.238,A -85,B 0,C 180,E1 -20648.495,E2 -20648.495} C_VEL
LIN {X 0,Y 235.579,Z 219.951,A -85,B 0,C 180,E1 -20650.212,E2 -20650.212} C_VEL
LIN {X 0,Y 230.373,Z 210.575,A -85,B 0,C 180,E1 -20652.314,E2 -20652.314} C_VEL
LIN {X 0,Y 226.226,Z 204.169,A -85,B 0,C 180,E1 -20654.096,E2 -20654.096} C_VEL
LIN {X 0,Y 223.242,Z 199.596,A -85,B 0,C 180,E1 -20655.494,E2 -20655.494} C_VEL
LIN {X 0,Y 219.215,Z 193.828,A -85,B 0,C 180,E1 -20657.541,E2 -20657.541} C_VEL
LIN {X 0,Y 215.77,Z 189.132,A -85,B 0,C 180,E1 -20659.503,E2 -20659.503} C_VEL
LIN {X 0,Y 215.363,Z 188.311,A -85,B 0,C 180,E1 -20659.87,E2 -20659.87} C_VEL
LIN {X 0,Y 214.693,Z 186.163,A -85,B 0,C 180,E1 -20661.776,E2 -20661.776} C_VEL
LIN {X 0,Y 213.762,Z 183.38,A -85,B 0,C 180,E1 -20665.081,E2 -20665.081} C_VEL
LIN {X 0,Y 213.761,Z 183.347,A -85,B 0,C 180,E1 -20668.735,E2 -20668.735} C_VEL
LIN {X 0,Y 213.78,Z 183.344,A -85,B 0,C 180,E1 -20672.596,E2 -20672.596} C_VEL
LIN {X 0,Y 213.791,Z 183.341,A -85,B 0,C 180,E1 -20676.985,E2 -20676.985} C_VEL
LIN {X 0,Y 213.875,Z 183.343,A -85,B 0,C 180,E1 -20682.797,E2 -20682.797} C_VEL
LIN {X 0,Y 213.913,Z 183.339,A -85,B 0,C 180,E1 -20686.703,E2 -20686.703} C_VEL
LIN {X 0,Y 214.125,Z 183.312,A -85,B 0,C 180,E1 -20690.554,E2 -20690.554} C_VEL
LIN {X 0,Y 214.071,Z 183.317,A -85,B 0,C 180,E1 -20694.347,E2 -20694.347} C_VEL
LIN {X 0,Y 214.396,Z 183.277,A -85,B 0,C 180,E1 -20698.121,E2 -20698.121} C_VEL
LIN {X 0,Y 214.423,Z 183.298,A -85,B 0,C 180,E1 -20701.643,E2 -20701.643} C_VEL
LIN {X 0,Y 214.489,Z 184.766,A -85,B 0,C 180,E1 -20703.286,E2 -20703.286} C_VEL
LIN {X 0,Y 215.029,Z 186.069,A -85,B 0,C 180,E1 -20704.158,E2 -20704.158} C_VEL
LIN {X 0,Y 218.59,Z 190.549,A -85,B 0,C 180,E1 -20706.228,E2 -20706.228} C_VEL
LIN {X 0,Y 219.921,Z 192.17,A -85,B 0,C 180,E1 -20706.931,E2 -20706.931} C_VEL
LIN {X 0,Y 223.878,Z 197.812,A -85,B 0,C 180,E1 -20708.916,E2 -20708.916} C_VEL
LIN {X 0,Y 227.547,Z 203.357,A -85,B 0,C 180,E1 -20710.606,E2 -20710.606} C_VEL
LIN {X 0,Y 231.052,Z 208.788,A -85,B 0,C 180,E1 -20712.084,E2 -20712.084} C_VEL
LIN {X 0,Y 236.253,Z 217.806,A -85,B 0,C 180,E1 -20714.15,E2 -20714.15} C_VEL
LIN {X 0,Y 242.532,Z 230.291,A -85,B 0,C 180,E1 -20716.438,E2 -20716.438} C_VEL
LIN {X 0,Y 245.998,Z 238.708,A -85,B 0,C 180,E1 -20717.68,E2 -20717.68} C_VEL
LIN {X 0,Y 242.432,Z 293.113,A -85,B 0,C 180,E1 -20719.435,E2 -20719.435} C_VEL
LIN {X 0,Y 240.65,Z 306.972,A -85,B 0,C 180,E1 -20720.183,E2 -20720.183} C_VEL
LIN {X 0,Y 238.472,Z 319.819,A -85,B 0,C 180,E1 -20721.255,E2 -20721.255} C_VEL
LIN {X 0,Y 235.525,Z 332.575,A -85,B 0,C 180,E1 -20722.685,E2 -20722.685} C_VEL
LIN {X 0,Y 232.418,Z 343.881,A -85,B 0,C 180,E1 -20724.371,E2 -20724.371} C_VEL
LIN {X 0,Y 229.193,Z 353.784,A -85,B 0,C 180,E1 -20726.249,E2 -20726.249} C_VEL
LIN {X 0,Y 225.739,Z 363.238,A -85,B 0,C 180,E1 -20728.515,E2 -20728.515} C_VEL
LIN {X 0,Y 222.793,Z 370.736,A -85,B 0,C 180,E1 -20730.779,E2 -20730.779} C_VEL
LIN {X 0,Y 219.551,Z 378.276,A -85,B 0,C 180,E1 -20733.671,E2 -20733.671} C_VEL
LIN {X 0,Y 217.379,Z 383.193,A -85,B 0,C 180,E1 -20736.078,E2 -20736.078} C_VEL
LIN {X 0,Y 215.564,Z 387.159,A -85,B 0,C 180,E1 -20738.517,E2 -20738.517} C_VEL
LIN {X 0,Y 213.432,Z 391.523,A -85,B 0,C 180,E1 -20742.246,E2 -20742.246} C_VEL
LIN {X 0,Y 212.103,Z 394.159,A -85,B 0,C 180,E1 -20745.91,E2 -20745.91} C_VEL
LIN {X 0,Y 211.516,Z 395.031,A -85,B 0,C 180,E1 -20748.357,E2 -20748.357} C_VEL
LIN {X 0,Y 211.124,Z 395.291,A -85,B 0,C 180,E1 -20750.77,E2 -20750.77} C_VEL
LIN {X 0,Y 210.935,Z 394.885,A -85,B 0,C 180,E1 -20753.153,E2 -20753.153} C_VEL
LIN {X 0,Y 210.972,Z 393.353,A -85,B 0,C 180,E1 -20756.387,E2 -20756.387} C_VEL
LIN {X 0,Y 211.511,Z 390.071,A -85,B 0,C 180,E1 -20760.108,E2 -20760.108} C_VEL
LIN {X 0,Y 212.233,Z 385.714,A -85,B 0,C 180,E1 -20763.39,E2 -20763.39} C_VEL
LIN {X 0,Y 213.299,Z 379.732,A -85,B 0,C 180,E1 -20766.712,E2 -20766.712} C_VEL
LIN {X 0,Y 214.564,Z 373.496,A -85,B 0,C 180,E1 -20769.386,E2 -20769.386} C_VEL
LIN {X 0,Y 216.11,Z 365.879,A -85,B 0,C 180,E1 -20772.007,E2 -20772.007} C_VEL
LIN {X 0,Y 218.115,Z 356.721,A -85,B 0,C 180,E1 -20774.526,E2 -20774.526} C_VEL
LIN {X 0,Y 220.031,Z 347.289,A -85,B 0,C 180,E1 -20776.613,E2 -20776.613} C_VEL
LIN {X 0,Y 221.933,Z 337.274,A -85,B 0,C 180,E1 -20778.386,E2 -20778.386} C_VEL
LIN {X 0,Y 223.799,Z 325.347,A -85,B 0,C 180,E1 -20780.056,E2 -20780.056} C_VEL
LIN {X 0,Y 225.477,Z 312.643,A -85,B 0,C 180,E1 -20781.402,E2 -20781.402} C_VEL
LIN {X 0,Y 226.789,Z 300.033,A -85,B 0,C 180,E1 -20782.343,E2 -20782.343} C_VEL
LIN {X 0,Y 227.74,Z 286.33,A -85,B 0,C 180,E1 -20783,E2 -20783} C_VEL
LIN {X 0,Y 230.247,Z 226.848,A -85,B 0,C 180,E1 -20784.979,E2 -20784.979} C_VEL
LIN {X 0,Y 229.369,Z 223.104,A -85,B 0,C 180,E1 -20785.223,E2 -20785.223} C_VEL
LIN {X 0,Y 222.519,Z 203.883,A -85,B 0,C 180,E1 -20786.805,E2 -20786.805} C_VEL
LIN {X 0,Y 214.705,Z 184.367,A -85,B 0,C 180,E1 -20788.712,E2 -20788.712} C_VEL
LIN {X 0,Y 214.5,Z 183.346,A -85,B 0,C 180,E1 -20789.181,E2 -20789.181} C_VEL
LIN {X 0,Y 214.443,Z 183.271,A -85,B 0,C 180,E1 -20791.88,E2 -20791.88} C_VEL
LIN {X 0,Y 214.192,Z 183.296,A -85,B 0,C 180,E1 -20797.543,E2 -20797.543} C_VEL
LIN {X 0,Y 213.995,Z 183.325,A -85,B 0,C 180,E1 -20801.366,E2 -20801.366} C_VEL
LIN {X 0,Y 213.929,Z 183.337,A -85,B 0,C 180,E1 -20805.239,E2 -20805.239} C_VEL
LIN {X 0,Y 213.839,Z 183.334,A -85,B 0,C 180,E1 -20809.189,E2 -20809.189} C_VEL
LIN {X 0,Y 213.848,Z 183.346,A -85,B 0,C 180,E1 -20813.229,E2 -20813.229} C_VEL
LIN {X 0,Y 213.83,Z 183.332,A -85,B 0,C 180,E1 -20817.452,E2 -20817.452} C_VEL
LIN {X 0,Y 213.768,Z 183.356,A -85,B 0,C 180,E1 -20821.739,E2 -20821.739} C_VEL
LIN {X 0,Y 213.744,Z 183.331,A -85,B 0,C 180,E1 -20826.29,E2 -20826.29} C_VEL
LIN {X 0,Y 213.714,Z 183.365,A -85,B 0,C 180,E1 -20831.127,E2 -20831.127} C_VEL
LIN {X 0,Y 213.709,Z 183.36,A -85,B 0,C 180,E1 -20833.68,E2 -20833.68} C_VEL
LIN {X 0,Y 213.708,Z 183.341,A -85,B 0,C 180,E1 -20836.345,E2 -20836.345} C_VEL
LIN {X 0,Y 213.719,Z 183.328,A -85,B 0,C 180,E1 -20839.144,E2 -20839.144} C_VEL
LIN {X 0,Y 213.743,Z 183.356,A -85,B 0,C 180,E1 -20843.713,E2 -20843.713} C_VEL
LIN {X 0,Y 213.761,Z 183.35,A -85,B 0,C 180,E1 -20848.262,E2 -20848.262} C_VEL
LIN {X 0,Y 213.791,Z 183.355,A -85,B 0,C 180,E1 -20852.599,E2 -20852.599} C_VEL
LIN {X 0,Y 213.814,Z 183.34,A -85,B 0,C 180,E1 -20856.98,E2 -20856.98} C_VEL
LIN {X 0,Y 213.947,Z 183.328,A -85,B 0,C 180,E1 -20862.805,E2 -20862.805} C_VEL
LIN {X 0,Y 213.954,Z 183.33,A -85,B 0,C 180,E1 -20866.707,E2 -20866.707} C_VEL
LIN {X 0,Y 214.137,Z 183.305,A -85,B 0,C 180,E1 -20870.556,E2 -20870.556} C_VEL
LIN {X 0,Y 214.076,Z 183.317,A -85,B 0,C 180,E1 -20874.349,E2 -20874.349} C_VEL
LIN {X 0,Y 214.409,Z 183.272,A -85,B 0,C 180,E1 -20878.122,E2 -20878.122} C_VEL
LIN {X 0,Y 214.515,Z 183.249,A -85,B 0,C 180,E1 -20880.001,E2 -20880.001} C_VEL
LIN {X 0,Y 214.409,Z 183.245,A -85,B 0,C 180,E1 -20881.879,E2 -20881.879} C_VEL
LIN {X 0,Y 214.188,Z 183.297,A -85,B 0,C 180,E1 -20887.543,E2 -20887.543} C_VEL
LIN {X 0,Y 213.998,Z 183.327,A -85,B 0,C 180,E1 -20891.365,E2 -20891.365} C_VEL
LIN {X 0,Y 213.901,Z 183.313,A -85,B 0,C 180,E1 -20895.24,E2 -20895.24} C_VEL
LIN {X 0,Y 213.797,Z 183.346,A -85,B 0,C 180,E1 -20899.192,E2 -20899.192} C_VEL
LIN {X 0,Y 213.769,Z 183.351,A -85,B 0,C 180,E1 -20903.237,E2 -20903.237} C_VEL
LIN {X 0,Y 213.79,Z 183.34,A -85,B 0,C 180,E1 -20907.427,E2 -20907.427} C_VEL
LIN {X 0,Y 213.764,Z 183.353,A -85,B 0,C 180,E1 -20911.739,E2 -20911.739} C_VEL
LIN {X 0,Y 213.747,Z 183.358,A -85,B 0,C 180,E1 -20916.289,E2 -20916.289} C_VEL
LIN {X 0,Y 213.703,Z 183.357,A -85,B 0,C 180,E1 -20921.128,E2 -20921.128} C_VEL
LIN {X 0,Y 213.706,Z 183.362,A -85,B 0,C 180,E1 -20923.68,E2 -20923.68} C_VEL
LIN {X 0,Y 213.706,Z 183.362,A -85,B 0,C 180,E1 -20926.345,E2 -20926.345} C_VEL
LIN {X 0,Y 213.687,Z 183.36,A -85,B 0,C 180,E1 -20930.461,E2 -20930.461} C_VEL
LIN {X 0,Y 213.294,Z 183.852,A -85,B 0,C 180,E1 -20931.389,E2 -20931.389} C_VEL
LIN {X 0,Y 211.923,Z 185.788,A -85,B 0,C 180,E1 -20932.577,E2 -20932.577} C_VEL
LIN {X 0,Y 210.308,Z 189.192,A -85,B 0,C 180,E1 -20933.751,E2 -20933.751} C_VEL
LIN {X 0,Y 209.762,Z 192.973,A -85,B 0,C 180,E1 -20934.593,E2 -20934.593} C_VEL
LIN {X 0,Y 210.451,Z 195.944,A -85,B 0,C 180,E1 -20935.022,E2 -20935.022} C_VEL
LIN {X 0,Y 218.274,Z 215.73,A -85,B 0,C 180,E1 -20936.914,E2 -20936.914} C_VEL
LIN {X 0,Y 221.293,Z 224.708,A -85,B 0,C 180,E1 -20937.655,E2 -20937.655} C_VEL
LIN {X 0,Y 223.385,Z 241.681,A -85,B 0,C 180,E1 -20938.582,E2 -20938.582} C_VEL
LIN {X 0,Y 220.809,Z 298.603,A -85,B 0,C 180,E1 -20940.569,E2 -20940.569} C_VEL
LIN {X 0,Y 219.439,Z 312.672,A -85,B 0,C 180,E1 -20941.417,E2 -20941.417} C_VEL
LIN {X 0,Y 217.957,Z 324.806,A -85,B 0,C 180,E1 -20942.514,E2 -20942.514} C_VEL
LIN {X 0,Y 216.1,Z 336.596,A -85,B 0,C 180,E1 -20943.955,E2 -20943.955} C_VEL
LIN {X 0,Y 214.218,Z 346.703,A -85,B 0,C 180,E1 -20945.529,E2 -20945.529} C_VEL
LIN {X 0,Y 212.146,Z 357.272,A -85,B 0,C 180,E1 -20947.604,E2 -20947.604} C_VEL
LIN {X 0,Y 210.308,Z 366.091,A -85,B 0,C 180,E1 -20949.762,E2 -20949.762} C_VEL
LIN {X 0,Y 208.418,Z 374.557,A -85,B 0,C 180,E1 -20952.331,E2 -20952.331} C_VEL
LIN {X 0,Y 206.724,Z 382.161,A -85,B 0,C 180,E1 -20955.226,E2 -20955.226} C_VEL
LIN {X 0,Y 205.577,Z 388.259,A -85,B 0,C 180,E1 -20958.162,E2 -20958.162} C_VEL
LIN {X 0,Y 204.819,Z 393.054,A -85,B 0,C 180,E1 -20961.115,E2 -20961.115} C_VEL
LIN {X 0,Y 204.407,Z 396.69,A -85,B 0,C 180,E1 -20964.078,E2 -20964.078} C_VEL
LIN {X 0,Y 204.299,Z 398.543,A -85,B 0,C 180,E1 -20966.053,E2 -20966.053} C_VEL
LIN {X 0,Y 204.29,Z 399.918,A -85,B 0,C 180,E1 -20968.026,E2 -20968.026} C_VEL
LIN {X 0,Y 204.377,Z 400.887,A -85,B 0,C 180,E1 -20969.998,E2 -20969.998} C_VEL
LIN {X 0,Y 204.29,Z 401.451,A -85,B 0,C 180,E1 -20971.969,E2 -20971.969} C_VEL
LIN {X 0,Y 204.323,Z 401.599,A -85,B 0,C 180,E1 -20974.042,E2 -20974.042} C_VEL
LIN {X 0,Y 204.498,Z 401.339,A -85,B 0,C 180,E1 -20975.916,E2 -20975.916} C_VEL
LIN {X 0,Y 205.201,Z 399.653,A -85,B 0,C 180,E1 -20979.858,E2 -20979.858} C_VEL
LIN {X 0,Y 205.875,Z 398.215,A -85,B 0,C 180,E1 -20981.817,E2 -20981.817} C_VEL
LIN {X 0,Y 207.232,Z 395.24,A -85,B 0,C 180,E1 -20984.733,E2 -20984.733} C_VEL
LIN {X 0,Y 209.113,Z 391.242,A -85,B 0,C 180,E1 -20987.604,E2 -20987.604} C_VEL
LIN {X 0,Y 212.176,Z 385.124,A -85,B 0,C 180,E1 -20990.857,E2 -20990.857} C_VEL
LIN {X 0,Y 215.324,Z 377.607,A -85,B 0,C 180,E1 -20993.949,E2 -20993.949} C_VEL
LIN {X 0,Y 218.38,Z 370.36,A -85,B 0,C 180,E1 -20996.261,E2 -20996.261} C_VEL
LIN {X 0,Y 221.608,Z 362.048,A -85,B 0,C 180,E1 -20998.403,E2 -20998.403} C_VEL
LIN {X 0,Y 225.253,Z 351.849,A -85,B 0,C 180,E1 -21000.462,E2 -21000.462} C_VEL
LIN {X 0,Y 228.756,Z 340.452,A -85,B 0,C 180,E1 -21002.26,E2 -21002.26} C_VEL
LIN {X 0,Y 231.707,Z 329.3,A -85,B 0,C 180,E1 -21003.608,E2 -21003.608} C_VEL
LIN {X 0,Y 234.318,Z 316.813,A -85,B 0,C 180,E1 -21004.739,E2 -21004.739} C_VEL
LIN {X 0,Y 236.413,Z 303.355,A -85,B 0,C 180,E1 -21005.601,E2 -21005.601} C_VEL
LIN {X 0,Y 237.729,Z 290.233,A -85,B 0,C 180,E1 -21006.12,E2 -21006.12} C_VEL
LIN {X 0,Y 240.616,Z 245.93,A -85,B 0,C 180,E1 -21007.559,E2 -21007.559} C_VEL
LIN {X 0,Y 239.996,Z 243.445,A -85,B 0,C 180,E1 -21007.836,E2 -21007.836} C_VEL
LIN {X 0,Y 235.797,Z 233.245,A -85,B 0,C 180,E1 -21009.45,E2 -21009.45} C_VEL
LIN {X 0,Y 231.126,Z 223.519,A -85,B 0,C 180,E1 -21011.342,E2 -21011.342} C_VEL
LIN {X 0,Y 226.353,Z 215.046,A -85,B 0,C 180,E1 -21013.375,E2 -21013.375} C_VEL
LIN {X 0,Y 222.813,Z 209.307,A -85,B 0,C 180,E1 -21015.024,E2 -21015.024} C_VEL
LIN {X 0,Y 220.092,Z 205.095,A -85,B 0,C 180,E1 -21016.365,E2 -21016.365} C_VEL
LIN {X 0,Y 216.564,Z 199.801,A -85,B 0,C 180,E1 -21018.276,E2 -21018.276} C_VEL
LIN {X 0,Y 213.172,Z 195.038,A -85,B 0,C 180,E1 -21020.299,E2 -21020.299} C_VEL
LIN {X 0,Y 208.082,Z 188.311,A -85,B 0,C 180,E1 -21023.932,E2 -21023.932} C_VEL
LIN {X 0,Y 207.731,Z 187.22,A -85,B 0,C 180,E1 -21024.889,E2 -21024.889} C_VEL
LIN {X 0,Y 206.692,Z 184.258,A -85,B 0,C 180,E1 -21029.296,E2 -21029.296} C_VEL
LIN {X 0,Y 206.696,Z 184.229,A -85,B 0,C 180,E1 -21033.766,E2 -21033.766} C_VEL
LIN {X 0,Y 206.708,Z 184.229,A -85,B 0,C 180,E1 -21038.037,E2 -21038.037} C_VEL
LIN {X 0,Y 206.794,Z 184.218,A -85,B 0,C 180,E1 -21042.189,E2 -21042.189} C_VEL
LIN {X 0,Y 206.854,Z 184.212,A -85,B 0,C 180,E1 -21046.241,E2 -21046.241} C_VEL
LIN {X 0,Y 207.07,Z 184.186,A -85,B 0,C 180,E1 -21050.229,E2 -21050.229} C_VEL
LIN {X 0,Y 207.034,Z 184.19,A -85,B 0,C 180,E1 -21054.154,E2 -21054.154} C_VEL
LIN {X 0,Y 207.361,Z 184.357,A -85,B 0,C 180,E1 -21058.057,E2 -21058.057} C_VEL
LIN {X 0,Y 207.978,Z 186.028,A -85,B 0,C 180,E1 -21060.06,E2 -21060.06} C_VEL
LIN {X 0,Y 209.641,Z 188.521,A -85,B 0,C 180,E1 -21061.44,E2 -21061.44} C_VEL
LIN {X 0,Y 213.3,Z 193.174,A -85,B 0,C 180,E1 -21063.896,E2 -21063.896} C_VEL
LIN {X 0,Y 216.538,Z 197.12,A -85,B 0,C 180,E1 -21065.794,E2 -21065.794} C_VEL
LIN {X 0,Y 220.94,Z 203.591,A -85,B 0,C 180,E1 -21068.157,E2 -21068.157} C_VEL
LIN {X 0,Y 224.525,Z 209.12,A -85,B 0,C 180,E1 -21069.884,E2 -21069.884} C_VEL
LIN {X 0,Y 228.702,Z 215.838,A -85,B 0,C 180,E1 -21071.738,E2 -21071.738} C_VEL
LIN {X 0,Y 234.565,Z 226.865,A -85,B 0,C 180,E1 -21074.15,E2 -21074.15} C_VEL
LIN {X 0,Y 239.057,Z 236.533,A -85,B 0,C 180,E1 -21075.864,E2 -21075.864} C_VEL
LIN {X 0,Y 240.918,Z 241.309,A -85,B 0,C 180,E1 -21076.573,E2 -21076.573} C_VEL
LIN {X 0,Y 237.275,Z 293.183,A -85,B 0,C 180,E1 -21078.269,E2 -21078.269} C_VEL
LIN {X 0,Y 235.415,Z 307.118,A -85,B 0,C 180,E1 -21079.035,E2 -21079.035} C_VEL
LIN {X 0,Y 233.17,Z 319.669,A -85,B 0,C 180,E1 -21080.091,E2 -21080.091} C_VEL
LIN {X 0,Y 230.222,Z 332.055,A -85,B 0,C 180,E1 -21081.488,E2 -21081.488} C_VEL
LIN {X 0,Y 227.128,Z 342.935,A -85,B 0,C 180,E1 -21083.094,E2 -21083.094} C_VEL
LIN {X 0,Y 223.473,Z 353.673,A -85,B 0,C 180,E1 -21085.128,E2 -21085.128} C_VEL
LIN {X 0,Y 219.825,Z 363.243,A -85,B 0,C 180,E1 -21087.457,E2 -21087.457} C_VEL
LIN {X 0,Y 216.631,Z 370.856,A -85,B 0,C 180,E1 -21089.798,E2 -21089.798} C_VEL
LIN {X 0,Y 213.167,Z 378.468,A -85,B 0,C 180,E1 -21092.807,E2 -21092.807} C_VEL
LIN {X 0,Y 210.702,Z 383.629,A -85,B 0,C 180,E1 -21095.438,E2 -21095.438} C_VEL
LIN {X 0,Y 208.047,Z 388.921,A -85,B 0,C 180,E1 -21099.021,E2 -21099.021} C_VEL
LIN {X 0,Y 206.627,Z 391.608,A -85,B 0,C 180,E1 -21101.562,E2 -21101.562} C_VEL
LIN {X 0,Y 205.544,Z 393.568,A -85,B 0,C 180,E1 -21104.111,E2 -21104.111} C_VEL
LIN {X 0,Y 204.81,Z 394.797,A -85,B 0,C 180,E1 -21106.666,E2 -21106.666} C_VEL
LIN {X 0,Y 204.249,Z 395.353,A -85,B 0,C 180,E1 -21109.199,E2 -21109.199} C_VEL
LIN {X 0,Y 203.848,Z 395.108,A -85,B 0,C 180,E1 -21112.462,E2 -21112.462} C_VEL
LIN {X 0,Y 203.867,Z 393.706,A -85,B 0,C 180,E1 -21115.827,E2 -21115.827} C_VEL
LIN {X 0,Y 204.239,Z 390.96,A -85,B 0,C 180,E1 -21119.345,E2 -21119.345} C_VEL
LIN {X 0,Y 204.848,Z 387.624,A -85,B 0,C 180,E1 -21122.224,E2 -21122.224} C_VEL
LIN {X 0,Y 205.879,Z 381.943,A -85,B 0,C 180,E1 -21125.821,E2 -21125.821} C_VEL
LIN {X 0,Y 207.286,Z 374.914,A -85,B 0,C 180,E1 -21129.148,E2 -21129.148} C_VEL
LIN {X 0,Y 208.903,Z 367.459,A -85,B 0,C 180,E1 -21131.918,E2 -21131.918} C_VEL
LIN {X 0,Y 210.852,Z 358.568,A -85,B 0,C 180,E1 -21134.537,E2 -21134.537} C_VEL
LIN {X 0,Y 212.974,Z 348.561,A -85,B 0,C 180,E1 -21136.889,E2 -21136.889} C_VEL
LIN {X 0,Y 215.143,Z 337.727,A -85,B 0,C 180,E1 -21138.905,E2 -21138.905} C_VEL
LIN {X 0,Y 216.892,Z 327.269,A -85,B 0,C 180,E1 -21140.443,E2 -21140.443} C_VEL
LIN {X 0,Y 218.685,Z 314.184,A -85,B 0,C 180,E1 -21141.919,E2 -21141.919} C_VEL
LIN {X 0,Y 220.105,Z 301.528,A -85,B 0,C 180,E1 -21142.938,E2 -21142.938} C_VEL
LIN {X 0,Y 221.152,Z 287.594,A -85,B 0,C 180,E1 -21143.652,E2 -21143.652} C_VEL
LIN {X 0,Y 223.713,Z 227.328,A -85,B 0,C 180,E1 -21145.728,E2 -21145.728} C_VEL
LIN {X 0,Y 217.09,Z 208.155,A -85,B 0,C 180,E1 -21147.335,E2 -21147.335} C_VEL
LIN {X 0,Y 208.328,Z 186.764,A -85,B 0,C 180,E1 -21149.456,E2 -21149.456} C_VEL
LIN {X 0,Y 207.612,Z 184.804,A -85,B 0,C 180,E1 -21149.76,E2 -21149.76} C_VEL
LIN {X 0,Y 207.495,Z 184.178,A -85,B 0,C 180,E1 -21150.245,E2 -21150.245} C_VEL
LIN {X 0,Y 207.078,Z 184.183,A -85,B 0,C 180,E1 -21153.894,E2 -21153.894} C_VEL
LIN {X 0,Y 207.135,Z 184.174,A -85,B 0,C 180,E1 -21157.802,E2 -21157.802} C_VEL
LIN {X 0,Y 206.919,Z 184.203,A -85,B 0,C 180,E1 -21161.761,E2 -21161.761} C_VEL
LIN {X 0,Y 206.864,Z 184.218,A -85,B 0,C 180,E1 -21165.773,E2 -21165.773} C_VEL
LIN {X 0,Y 206.784,Z 184.215,A -85,B 0,C 180,E1 -21169.871,E2 -21169.871} C_VEL
LIN {X 0,Y 206.764,Z 184.225,A -85,B 0,C 180,E1 -21174.074,E2 -21174.074} C_VEL
LIN {X 0,Y 206.737,Z 184.224,A -85,B 0,C 180,E1 -21178.422,E2 -21178.422} C_VEL
LIN {X 0,Y 206.699,Z 184.231,A -85,B 0,C 180,E1 -21182.959,E2 -21182.959} C_VEL
LIN {X 0,Y 206.68,Z 184.218,A -85,B 0,C 180,E1 -21187.742,E2 -21187.742} C_VEL
LIN {X 0,Y 206.644,Z 184.244,A -85,B 0,C 180,E1 -21191.565,E2 -21191.565} C_VEL
LIN {X 0,Y 206.636,Z 184.23,A -85,B 0,C 180,E1 -21195.583,E2 -21195.583} C_VEL
LIN {X 0,Y 206.662,Z 184.21,A -85,B 0,C 180,E1 -21199.75,E2 -21199.75} C_VEL
LIN {X 0,Y 206.702,Z 184.238,A -85,B 0,C 180,E1 -21204.69,E2 -21204.69} C_VEL
LIN {X 0,Y 206.698,Z 184.227,A -85,B 0,C 180,E1 -21209.336,E2 -21209.336} C_VEL
LIN {X 0,Y 206.708,Z 184.236,A -85,B 0,C 180,E1 -21213.77,E2 -21213.77} C_VEL
LIN {X 0,Y 206.74,Z 184.223,A -85,B 0,C 180,E1 -21218.042,E2 -21218.042} C_VEL
LIN {X 0,Y 206.876,Z 184.212,A -85,B 0,C 180,E1 -21222.198,E2 -21222.198} C_VEL
LIN {X 0,Y 206.896,Z 184.206,A -85,B 0,C 180,E1 -21226.245,E2 -21226.245} C_VEL
LIN {X 0,Y 207.082,Z 184.185,A -85,B 0,C 180,E1 -21230.231,E2 -21230.231} C_VEL
LIN {X 0,Y 207.04,Z 184.191,A -85,B 0,C 180,E1 -21234.156,E2 -21234.156} C_VEL
LIN {X 0,Y 207.348,Z 184.152,A -85,B 0,C 180,E1 -21238.058,E2 -21238.058} C_VEL
LIN {X 0,Y 207.483,Z 184.124,A -85,B 0,C 180,E1 -21240.001,E2 -21240.001} C_VEL
LIN {X 0,Y 207.348,Z 184.123,A -85,B 0,C 180,E1 -21241.943,E2 -21241.943} C_VEL
LIN {X 0,Y 207.133,Z 184.178,A -85,B 0,C 180,E1 -21247.801,E2 -21247.801} C_VEL
LIN {X 0,Y 206.92,Z 184.205,A -85,B 0,C 180,E1 -21251.759,E2 -21251.759} C_VEL
LIN {X 0,Y 206.827,Z 184.191,A -85,B 0,C 180,E1 -21255.775,E2 -21255.775} C_VEL
LIN {X 0,Y 206.718,Z 184.234,A -85,B 0,C 180,E1 -21259.877,E2 -21259.877} C_VEL
LIN {X 0,Y 206.696,Z 184.228,A -85,B 0,C 180,E1 -21264.081,E2 -21264.081} C_VEL
LIN {X 0,Y 206.692,Z 184.233,A -85,B 0,C 180,E1 -21268.427,E2 -21268.427} C_VEL
LIN {X 0,Y 206.699,Z 184.223,A -85,B 0,C 180,E1 -21272.958,E2 -21272.958} C_VEL
LIN {X 0,Y 206.673,Z 184.24,A -85,B 0,C 180,E1 -21277.742,E2 -21277.742} C_VEL
LIN {X 0,Y 206.636,Z 184.241,A -85,B 0,C 180,E1 -21281.559,E2 -21281.559} C_VEL
LIN {X 0,Y 206.635,Z 184.237,A -85,B 0,C 180,E1 -21285.583,E2 -21285.583} C_VEL
LIN {X 0,Y 206.677,Z 184.238,A -85,B 0,C 180,E1 -21290.684,E2 -21290.684} C_VEL
LIN {X 0,Y 206.759,Z 184.527,A -85,B 0,C 180,E1 -21291.622,E2 -21291.622} C_VEL
LIN {X 0,Y 208.048,Z 190.143,A -85,B 0,C 180,E1 -21294.368,E2 -21294.368} C_VEL
LIN {X 0,Y 210.451,Z 195.944,A -85,B 0,C 180,E1 -21295.022,E2 -21295.022} C_VEL
LIN {X 0,Y 212.254,Z 201.27,A -85,B 0,C 180,E1 -21295.502,E2 -21295.502} C_VEL
LIN {X 0,Y 213.729,Z 210.763,A -85,B 0,C 180,E1 -21296.104,E2 -21296.104} C_VEL
LIN {X 0,Y 214.988,Z 226.436,A -85,B 0,C 180,E1 -21296.924,E2 -21296.924} C_VEL
LIN {X 0,Y 216.927,Z 242.619,A -85,B 0,C 180,E1 -21297.832,E2 -21297.832} C_VEL
LIN {X 0,Y 214.28,Z 298.721,A -85,B 0,C 180,E1 -21299.851,E2 -21299.851} C_VEL
LIN {X 0,Y 212.85,Z 312.684,A -85,B 0,C 180,E1 -21300.718,E2 -21300.718} C_VEL
LIN {X 0,Y 211.322,Z 324.774,A -85,B 0,C 180,E1 -21301.845,E2 -21301.845} C_VEL
LIN {X 0,Y 209.412,Z 336.544,A -85,B 0,C 180,E1 -21303.327,E2 -21303.327} C_VEL
LIN {X 0,Y 207.468,Z 346.636,A -85,B 0,C 180,E1 -21304.946,E2 -21304.946} C_VEL
LIN {X 0,Y 205.323,Z 357.196,A -85,B 0,C 180,E1 -21307.084,E2 -21307.084} C_VEL
LIN {X 0,Y 203.377,Z 366.128,A -85,B 0,C 180,E1 -21309.342,E2 -21309.342} C_VEL
LIN {X 0,Y 201.331,Z 375.159,A -85,B 0,C 180,E1 -21312.213,E2 -21312.213} C_VEL
LIN {X 0,Y 199.602,Z 382.634,A -85,B 0,C 180,E1 -21315.208,E2 -21315.208} C_VEL
LIN {X 0,Y 198.599,Z 387.697,A -85,B 0,C 180,E1 -21317.739,E2 -21317.739} C_VEL
LIN {X 0,Y 197.796,Z 392.587,A -85,B 0,C 180,E1 -21320.797,E2 -21320.797} C_VEL
LIN {X 0,Y 197.345,Z 396.31,A -85,B 0,C 180,E1 -21323.865,E2 -21323.865} C_VEL
LIN {X 0,Y 197.186,Z 398.565,A -85,B 0,C 180,E1 -21326.355,E2 -21326.355} C_VEL
LIN {X 0,Y 197.281,Z 400.671,A -85,B 0,C 180,E1 -21329.998,E2 -21329.998} C_VEL
LIN {X 0,Y 197.241,Z 401.482,A -85,B 0,C 180,E1 -21333.89,E2 -21333.89} C_VEL
LIN {X 0,Y 197.413,Z 401.289,A -85,B 0,C 180,E1 -21336.129,E2 -21336.129} C_VEL
LIN {X 0,Y 198.198,Z 399.684,A -85,B 0,C 180,E1 -21340.21,E2 -21340.21} C_VEL
LIN {X 0,Y 198.925,Z 398.299,A -85,B 0,C 180,E1 -21342.236,E2 -21342.236} C_VEL
LIN {X 0,Y 200.352,Z 395.407,A -85,B 0,C 180,E1 -21345.251,E2 -21345.251} C_VEL
LIN {X 0,Y 202.376,Z 391.515,A -85,B 0,C 180,E1 -21348.21,E2 -21348.21} C_VEL
LIN {X 0,Y 205.069,Z 386.515,A -85,B 0,C 180,E1 -21351.088,E2 -21351.088} C_VEL
LIN {X 0,Y 207.887,Z 380.293,A -85,B 0,C 180,E1 -21353.931,E2 -21353.931} C_VEL
LIN {X 0,Y 211.433,Z 372.541,A -85,B 0,C 180,E1 -21356.66,E2 -21356.66} C_VEL
LIN {X 0,Y 215.446,Z 362.909,A -85,B 0,C 180,E1 -21359.293,E2 -21359.293} C_VEL
LIN {X 0,Y 219.234,Z 353.027,A -85,B 0,C 180,E1 -21361.392,E2 -21361.392} C_VEL
LIN {X 0,Y 222.859,Z 341.971,A -85,B 0,C 180,E1 -21363.222,E2 -21363.222} C_VEL
LIN {X 0,Y 226.368,Z 329.537,A -85,B 0,C 180,E1 -21364.781,E2 -21364.781} C_VEL
LIN {X 0,Y 229.09,Z 317.254,A -85,B 0,C 180,E1 -21365.921,E2 -21365.921} C_VEL
LIN {X 0,Y 231.305,Z 303.731,A -85,B 0,C 180,E1 -21366.805,E2 -21366.805} C_VEL
LIN {X 0,Y 232.715,Z 290.65,A -85,B 0,C 180,E1 -21367.335,E2 -21367.335} C_VEL
LIN {X 0,Y 235.632,Z 247.527,A -85,B 0,C 180,E1 -21368.759,E2 -21368.759} C_VEL
LIN {X 0,Y 231.635,Z 237.476,A -85,B 0,C 180,E1 -21370.412,E2 -21370.412} C_VEL
LIN {X 0,Y 227.286,Z 228.207,A -85,B 0,C 180,E1 -21372.281,E2 -21372.281} C_VEL
LIN {X 0,Y 222.951,Z 220.265,A -85,B 0,C 180,E1 -21374.264,E2 -21374.264} C_VEL
LIN {X 0,Y 219.892,Z 215.125,A -85,B 0,C 180,E1 -21375.766,E2 -21375.766} C_VEL
LIN {X 0,Y 217.26,Z 210.88,A -85,B 0,C 180,E1 -21377.143,E2 -21377.143} C_VEL
LIN {X 0,Y 214.088,Z 205.964,A -85,B 0,C 180,E1 -21378.961,E2 -21378.961} C_VEL
LIN {X 0,Y 210.008,Z 200.167,A -85,B 0,C 180,E1 -21381.558,E2 -21381.558} C_VEL
LIN {X 0,Y 205.348,Z 193.89,A -85,B 0,C 180,E1 -21385.126,E2 -21385.126} C_VEL
LIN {X 0,Y 201.697,Z 189.53,A -85,B 0,C 180,E1 -21388.634,E2 -21388.634} C_VEL
LIN {X 0,Y 200.371,Z 187.511,A -85,B 0,C 180,E1 -21390.589,E2 -21390.589} C_VEL
LIN {X 0,Y 199.694,Z 185.366,A -85,B 0,C 180,E1 -21395.017,E2 -21395.017} C_VEL
LIN {X 0,Y 199.67,Z 185.101,A -85,B 0,C 180,E1 -21397.22,E2 -21397.22} C_VEL
LIN {X 0,Y 199.737,Z 185.093,A -85,B 0,C 180,E1 -21401.801,E2 -21401.801} C_VEL
LIN {X 0,Y 199.792,Z 185.086,A -85,B 0,C 180,E1 -21405.744,E2 -21405.744} C_VEL
LIN {X 0,Y 200.048,Z 185.105,A -85,B 0,C 180,E1 -21410.903,E2 -21410.903} C_VEL
LIN {X 0,Y 200.163,Z 185.869,A -85,B 0,C 180,E1 -21412.94,E2 -21412.94} C_VEL
LIN {X 0,Y 200.623,Z 187.216,A -85,B 0,C 180,E1 -21414.219,E2 -21414.219} C_VEL
LIN {X 0,Y 202.398,Z 189.533,A -85,B 0,C 180,E1 -21416.291,E2 -21416.291} C_VEL
LIN {X 0,Y 204.858,Z 191.353,A -85,B 0,C 180,E1 -21418.525,E2 -21418.525} C_VEL
LIN {X 0,Y 206.169,Z 192.951,A -85,B 0,C 180,E1 -21419.633,E2 -21419.633} C_VEL
LIN {X 0,Y 210.976,Z 199.351,A -85,B 0,C 180,E1 -21423.191,E2 -21423.191} C_VEL
LIN {X 0,Y 214.245,Z 203.483,A -85,B 0,C 180,E1 -21425.204,E2 -21425.204} C_VEL
LIN {X 0,Y 218.55,Z 210.147,A -85,B 0,C 180,E1 -21427.641,E2 -21427.641} C_VEL
LIN {X 0,Y 223.542,Z 218.133,A -85,B 0,C 180,E1 -21430.099,E2 -21430.099} C_VEL
LIN {X 0,Y 228.775,Z 227.692,A -85,B 0,C 180,E1 -21432.448,E2 -21432.448} C_VEL
LIN {X 0,Y 234.235,Z 239.385,A -85,B 0,C 180,E1 -21434.728,E2 -21434.728} C_VEL
LIN {X 0,Y 235.88,Z 243.543,A -85,B 0,C 180,E1 -21435.388,E2 -21435.388} C_VEL
LIN {X 0,Y 232.232,Z 293.587,A -85,B 0,C 180,E1 -21437.057,E2 -21437.057} C_VEL
LIN {X 0,Y 230.322,Z 307.279,A -85,B 0,C 180,E1 -21437.817,E2 -21437.817} C_VEL
LIN {X 0,Y 227.999,Z 319.746,A -85,B 0,C 180,E1 -21438.878,E2 -21438.878} C_VEL
LIN {X 0,Y 224.821,Z 332.381,A -85,B 0,C 180,E1 -21440.32,E2 -21440.32} C_VEL
LIN {X 0,Y 221.605,Z 343.121,A -85,B 0,C 180,E1 -21441.938,E2 -21441.938} C_VEL
LIN {X 0,Y 218.026,Z 353.126,A -85,B 0,C 180,E1 -21443.849,E2 -21443.849} C_VEL
LIN {X 0,Y 213.85,Z 363.566,A -85,B 0,C 180,E1 -21446.427,E2 -21446.427} C_VEL
LIN {X 0,Y 210.498,Z 371.083,A -85,B 0,C 180,E1 -21448.792,E2 -21448.792} C_VEL
LIN {X 0,Y 206.87,Z 378.648,A -85,B 0,C 180,E1 -21451.867,E2 -21451.867} C_VEL
LIN {X 0,Y 203.591,Z 385.008,A -85,B 0,C 180,E1 -21455.299,E2 -21455.299} C_VEL
LIN {X 0,Y 201.496,Z 388.839,A -85,B 0,C 180,E1 -21458.073,E2 -21458.073} C_VEL
LIN {X 0,Y 199.247,Z 392.718,A -85,B 0,C 180,E1 -21462.08,E2 -21462.08} C_VEL
LIN {X 0,Y 198.069,Z 394.558,A -85,B 0,C 180,E1 -21465.205,E2 -21465.205} C_VEL
LIN {X 0,Y 197.272,Z 395.447,A -85,B 0,C 180,E1 -21468.429,E2 -21468.429} C_VEL
LIN {X 0,Y 196.822,Z 395.315,A -85,B 0,C 180,E1 -21471.771,E2 -21471.771} C_VEL
LIN {X 0,Y 196.749,Z 394.04,A -85,B 0,C 180,E1 -21475.241,E2 -21475.241} C_VEL
LIN {X 0,Y 197.064,Z 391.443,A -85,B 0,C 180,E1 -21478.86,E2 -21478.86} C_VEL
LIN {X 0,Y 197.585,Z 388.923,A -85,B 0,C 180,E1 -21481.305,E2 -21481.305} C_VEL
LIN {X 0,Y 198.441,Z 383.968,A -85,B 0,C 180,E1 -21484.853,E2 -21484.853} C_VEL
LIN {X 0,Y 199.734,Z 377.518,A -85,B 0,C 180,E1 -21488.32,E2 -21488.32} C_VEL
LIN {X 0,Y 201.268,Z 370.531,A -85,B 0,C 180,E1 -21491.234,E2 -21491.234} C_VEL
LIN {X 0,Y 203.184,Z 362.386,A -85,B 0,C 180,E1 -21493.938,E2 -21493.938} C_VEL
LIN {X 0,Y 205.419,Z 352.156,A -85,B 0,C 180,E1 -21496.65,E2 -21496.65} C_VEL
LIN {X 0,Y 207.709,Z 341.348,A -85,B 0,C 180,E1 -21498.879,E2 -21498.879} C_VEL
LIN {X 0,Y 209.917,Z 329.108,A -85,B 0,C 180,E1 -21500.852,E2 -21500.852} C_VEL
LIN {X 0,Y 211.684,Z 317.719,A -85,B 0,C 180,E1 -21502.251,E2 -21502.251} C_VEL
LIN {X 0,Y 213.208,Z 304.331,A -85,B 0,C 180,E1 -21503.461,E2 -21503.461} C_VEL
LIN {X 0,Y 214.477,Z 290.881,A -85,B 0,C 180,E1 -21504.253,E2 -21504.253} C_VEL
LIN {X 0,Y 217.231,Z 228.589,A -85,B 0,C 180,E1 -21506.484,E2 -21506.484} C_VEL
LIN {X 0,Y 210.513,Z 209.436,A -85,B 0,C 180,E1 -21508.168,E2 -21508.168} C_VEL
LIN {X 0,Y 202.709,Z 190.354,A -85,B 0,C 180,E1 -21510.141,E2 -21510.141} C_VEL
LIN {X 0,Y 200.551,Z 185.879,A -85,B 0,C 180,E1 -21510.755,E2 -21510.755} C_VEL
LIN {X 0,Y 200.377,Z 185.093,A -85,B 0,C 180,E1 -21511.195,E2 -21511.195} C_VEL
LIN {X 0,Y 200.084,Z 185.052,A -85,B 0,C 180,E1 -21518.079,E2 -21518.079} C_VEL
LIN {X 0,Y 199.87,Z 185.077,A -85,B 0,C 180,E1 -21522.182,E2 -21522.182} C_VEL
LIN {X 0,Y 199.803,Z 185.096,A -85,B 0,C 180,E1 -21526.346,E2 -21526.346} C_VEL
LIN {X 0,Y 199.7,Z 185.103,A -85,B 0,C 180,E1 -21530.607,E2 -21530.607} C_VEL
LIN {X 0,Y 199.673,Z 185.097,A -85,B 0,C 180,E1 -21534.986,E2 -21534.986} C_VEL
LIN {X 0,Y 199.665,Z 185.111,A -85,B 0,C 180,E1 -21539.526,E2 -21539.526} C_VEL
LIN {X 0,Y 199.672,Z 185.112,A -85,B 0,C 180,E1 -21542.357,E2 -21542.357} C_VEL
LIN {X 0,Y 199.623,Z 185.088,A -85,B 0,C 180,E1 -21546.765,E2 -21546.765} C_VEL
LIN {X 0,Y 199.609,Z 185.111,A -85,B 0,C 180,E1 -21549.33,E2 -21549.33} C_VEL
LIN {X 0,Y 199.577,Z 185.125,A -85,B 0,C 180,E1 -21552.312,E2 -21552.312} C_VEL
LIN {X 0,Y 199.582,Z 185.11,A -85,B 0,C 180,E1 -21555.231,E2 -21555.231} C_VEL
LIN {X 0,Y 199.581,Z 185.084,A -85,B 0,C 180,E1 -21558.007,E2 -21558.007} C_VEL
LIN {X 0,Y 199.609,Z 185.095,A -85,B 0,C 180,E1 -21560.77,E2 -21560.77} C_VEL
LIN {X 0,Y 199.612,Z 185.119,A -85,B 0,C 180,E1 -21565.715,E2 -21565.715} C_VEL
LIN {X 0,Y 199.688,Z 185.103,A -85,B 0,C 180,E1 -21568.136,E2 -21568.136} C_VEL
LIN {X 0,Y 199.646,Z 185.116,A -85,B 0,C 180,E1 -21572.767,E2 -21572.767} C_VEL
LIN {X 0,Y 199.712,Z 185.096,A -85,B 0,C 180,E1 -21577.227,E2 -21577.227} C_VEL
LIN {X 0,Y 199.8,Z 185.096,A -85,B 0,C 180,E1 -21581.759,E2 -21581.759} C_VEL
LIN {X 0,Y 199.837,Z 185.082,A -85,B 0,C 180,E1 -21585.749,E2 -21585.749} C_VEL
LIN {X 0,Y 200.027,Z 185.066,A -85,B 0,C 180,E1 -21589.883,E2 -21589.883} C_VEL
LIN {X 0,Y 200.004,Z 185.065,A -85,B 0,C 180,E1 -21593.95,E2 -21593.95} C_VEL
LIN {X 0,Y 200.29,Z 185.031,A -85,B 0,C 180,E1 -21597.99,E2 -21597.99} C_VEL
LIN {X 0,Y 200.451,Z 184.999,A -85,B 0,C 180,E1 -21600.001,E2 -21600.001} C_VEL
LIN {X 0,Y 199.993,Z 185.033,A -85,B 0,C 180,E1 -21604.031,E2 -21604.031} C_VEL
LIN {X 0,Y 200.08,Z 185.058,A -85,B 0,C 180,E1 -21608.078,E2 -21608.078} C_VEL
LIN {X 0,Y 199.869,Z 185.082,A -85,B 0,C 180,E1 -21612.181,E2 -21612.181} C_VEL
LIN {X 0,Y 199.76,Z 185.07,A -85,B 0,C 180,E1 -21616.348,E2 -21616.348} C_VEL
LIN {X 0,Y 199.648,Z 185.115,A -85,B 0,C 180,E1 -21620.612,E2 -21620.612} C_VEL
LIN {X 0,Y 199.626,Z 185.098,A -85,B 0,C 180,E1 -21624.992,E2 -21624.992} C_VEL
LIN {X 0,Y 199.613,Z 185.122,A -85,B 0,C 180,E1 -21629.533,E2 -21629.533} C_VEL
LIN {X 0,Y 199.671,Z 185.103,A -85,B 0,C 180,E1 -21632.352,E2 -21632.352} C_VEL
LIN {X 0,Y 199.623,Z 185.119,A -85,B 0,C 180,E1 -21636.764,E2 -21636.764} C_VEL
LIN {X 0,Y 199.6,Z 185.11,A -85,B 0,C 180,E1 -21639.331,E2 -21639.331} C_VEL
LIN {X 0,Y 199.571,Z 185.125,A -85,B 0,C 180,E1 -21642.307,E2 -21642.307} C_VEL
LIN {X 0,Y 199.581,Z 185.114,A -85,B 0,C 180,E1 -21645.227,E2 -21645.227} C_VEL
LIN {X 0,Y 199.663,Z 185.228,A -85,B 0,C 180,E1 -21650.751,E2 -21650.751} C_VEL
LIN {X 0,Y 200.756,Z 189.936,A -85,B 0,C 180,E1 -21653.232,E2 -21653.232} C_VEL
LIN {X 0,Y 203.726,Z 196.943,A -85,B 0,C 180,E1 -21654.089,E2 -21654.089} C_VEL
LIN {X 0,Y 211.694,Z 217.047,A -85,B 0,C 180,E1 -21656.097,E2 -21656.097} C_VEL
LIN {X 0,Y 214.988,Z 226.436,A -85,B 0,C 180,E1 -21656.924,E2 -21656.924} C_VEL
LIN {X 0,Y 215.044,Z 232.271,A -85,B 0,C 180,E1 -21657.173,E2 -21657.173} C_VEL
LIN {X 0,Y 214.058,Z 238.133,A -85,B 0,C 180,E1 -21657.291,E2 -21657.291} C_VEL
LIN {X 0,Y 210.215,Z 253.761,A -85,B 0,C 180,E1 -21657.455,E2 -21657.455} C_VEL
LIN {X 0,Y 209.802,Z 257.738,A -85,B 0,C 180,E1 -21657.569,E2 -21657.569} C_VEL
LIN {X 0,Y 207.723,Z 299.067,A -85,B 0,C 180,E1 -21659.121,E2 -21659.121} C_VEL
LIN {X 0,Y 206.297,Z 312.423,A -85,B 0,C 180,E1 -21659.974,E2 -21659.974} C_VEL
LIN {X 0,Y 204.719,Z 324.56,A -85,B 0,C 180,E1 -21661.132,E2 -21661.132} C_VEL
LIN {X 0,Y 202.741,Z 336.351,A -85,B 0,C 180,E1 -21662.656,E2 -21662.656} C_VEL
LIN {X 0,Y 200.742,Z 346.461,A -85,B 0,C 180,E1 -21664.324,E2 -21664.324} C_VEL
LIN {X 0,Y 198.518,Z 357.034,A -85,B 0,C 180,E1 -21666.528,E2 -21666.528} C_VEL
LIN {X 0,Y 196.375,Z 366.544,A -85,B 0,C 180,E1 -21669.028,E2 -21669.028} C_VEL
LIN {X 0,Y 194.222,Z 375.71,A -85,B 0,C 180,E1 -21672.085,E2 -21672.085} C_VEL
LIN {X 0,Y 192.435,Z 383.067,A -85,B 0,C 180,E1 -21675.186,E2 -21675.186} C_VEL
LIN {X 0,Y 191.284,Z 388.934,A -85,B 0,C 180,E1 -21678.34,E2 -21678.34} C_VEL
LIN {X 0,Y 190.547,Z 393.518,A -85,B 0,C 180,E1 -21681.514,E2 -21681.514} C_VEL
LIN {X 0,Y 190.283,Z 395.921,A -85,B 0,C 180,E1 -21683.636,E2 -21683.636} C_VEL
LIN {X 0,Y 190.092,Z 398.531,A -85,B 0,C 180,E1 -21686.605,E2 -21686.605} C_VEL
LIN {X 0,Y 190.187,Z 400.456,A -85,B 0,C 180,E1 -21689.998,E2 -21689.998} C_VEL
LIN {X 0,Y 190.118,Z 401.317,A -85,B 0,C 180,E1 -21693.522,E2 -21693.522} C_VEL
LIN {X 0,Y 190.357,Z 401.23,A -85,B 0,C 180,E1 -21696.357,E2 -21696.357} C_VEL
LIN {X 0,Y 191.214,Z 399.724,A -85,B 0,C 180,E1 -21700.587,E2 -21700.587} C_VEL
LIN {X 0,Y 192.956,Z 396.657,A -85,B 0,C 180,E1 -21704.769,E2 -21704.769} C_VEL
LIN {X 0,Y 194.817,Z 393.206,A -85,B 0,C 180,E1 -21707.854,E2 -21707.854} C_VEL
LIN {X 0,Y 197.468,Z 388.69,A -85,B 0,C 180,E1 -21710.846,E2 -21710.846} C_VEL
LIN {X 0,Y 200.451,Z 383.007,A -85,B 0,C 180,E1 -21713.776,E2 -21713.776} C_VEL
LIN {X 0,Y 203.859,Z 375.953,A -85,B 0,C 180,E1 -21716.624,E2 -21716.624} C_VEL
LIN {X 0,Y 207.949,Z 367.216,A -85,B 0,C 180,E1 -21719.341,E2 -21719.341} C_VEL
LIN {X 0,Y 211.729,Z 358.311,A -85,B 0,C 180,E1 -21721.517,E2 -21721.517} C_VEL
LIN {X 0,Y 215.381,Z 348.582,A -85,B 0,C 180,E1 -21723.408,E2 -21723.408} C_VEL
LIN {X 0,Y 218.871,Z 337.899,A -85,B 0,C 180,E1 -21725.025,E2 -21725.025} C_VEL
LIN {X 0,Y 222.076,Z 326.098,A -85,B 0,C 180,E1 -21726.394,E2 -21726.394} C_VEL
LIN {X 0,Y 224.711,Z 313.987,A -85,B 0,C 180,E1 -21727.436,E2 -21727.436} C_VEL
LIN {X 0,Y 226.783,Z 300.736,A -85,B 0,C 180,E1 -21728.228,E2 -21728.228} C_VEL
LIN {X 0,Y 228.443,Z 282.334,A -85,B 0,C 180,E1 -21728.894,E2 -21728.894} C_VEL
LIN {X 0,Y 230.794,Z 250.619,A -85,B 0,C 180,E1 -21729.94,E2 -21729.94} C_VEL
LIN {X 0,Y 230.294,Z 248.581,A -85,B 0,C 180,E1 -21730.198,E2 -21730.198} C_VEL
LIN {X 0,Y 225.758,Z 237.525,A -85,B 0,C 180,E1 -21732.228,E2 -21732.228} C_VEL
LIN {X 0,Y 221.263,Z 228.457,A -85,B 0,C 180,E1 -21734.357,E2 -21734.357} C_VEL
LIN {X 0,Y 216.858,Z 220.713,A -85,B 0,C 180,E1 -21736.602,E2 -21736.602} C_VEL
LIN {X 0,Y 214.184,Z 216.206,A -85,B 0,C 180,E1 -21738.128,E2 -21738.128} C_VEL
LIN {X 0,Y 211.388,Z 211.792,A -85,B 0,C 180,E1 -21739.818,E2 -21739.818} C_VEL
LIN {X 0,Y 207.803,Z 206.423,A -85,B 0,C 180,E1 -21742.261,E2 -21742.261} C_VEL
LIN {X 0,Y 203.542,Z 200.455,A -85,B 0,C 180,E1 -21745.694,E2 -21745.694} C_VEL
LIN {X 0,Y 200.065,Z 196.111,A -85,B 0,C 180,E1 -21749.231,E2 -21749.231} C_VEL
LIN {X 0,Y 198.245,Z 193.804,A -85,B 0,C 180,E1 -21751.622,E2 -21751.622} C_VEL
LIN {X 0,Y 195.715,Z 191.004,A -85,B 0,C 180,E1 -21756.392,E2 -21756.392} C_VEL
LIN {X 0,Y 194.652,Z 190.118,A -85,B 0,C 180,E1 -21761.037,E2 -21761.037} C_VEL
LIN {X 0,Y 195.086,Z 190.378,A -85,B 0,C 180,E1 -21765.925,E2 -21765.925} C_VEL
LIN {X 0,Y 197.86,Z 192.047,A -85,B 0,C 180,E1 -21771.831,E2 -21771.831} C_VEL
LIN {X 0,Y 198.9,Z 193.524,A -85,B 0,C 180,E1 -21773.404,E2 -21773.404} C_VEL
LIN {X 0,Y 200.76,Z 196.214,A -85,B 0,C 180,E1 -21775.733,E2 -21775.733} C_VEL
LIN {X 0,Y 203.259,Z 198.091,A -85,B 0,C 180,E1 -21778.095,E2 -21778.095} C_VEL
LIN {X 0,Y 204.406,Z 199.677,A -85,B 0,C 180,E1 -21779.137,E2 -21779.137} C_VEL
LIN {X 0,Y 208.775,Z 205.647,A -85,B 0,C 180,E1 -21782.519,E2 -21782.519} C_VEL
LIN {X 0,Y 212.351,Z 210.617,A -85,B 0,C 180,E1 -21784.849,E2 -21784.849} C_VEL
LIN {X 0,Y 215.706,Z 215.874,A -85,B 0,C 180,E1 -21786.823,E2 -21786.823} C_VEL
LIN {X 0,Y 220.298,Z 223.46,A -85,B 0,C 180,E1 -21789.236,E2 -21789.236} C_VEL
LIN {X 0,Y 225.539,Z 233.542,A -85,B 0,C 180,E1 -21791.752,E2 -21791.752} C_VEL
LIN {X 0,Y 230.316,Z 244.162,A -85,B 0,C 180,E1 -21793.849,E2 -21793.849} C_VEL
LIN {X 0,Y 231.048,Z 246.206,A -85,B 0,C 180,E1 -21794.178,E2 -21794.178} C_VEL
LIN {X 0,Y 227.36,Z 293.574,A -85,B 0,C 180,E1 -21795.773,E2 -21795.773} C_VEL
LIN {X 0,Y 225.409,Z 307.073,A -85,B 0,C 180,E1 -21796.524,E2 -21796.524} C_VEL
LIN {X 0,Y 222.984,Z 319.489,A -85,B 0,C 180,E1 -21797.566,E2 -21797.566} C_VEL
LIN {X 0,Y 219.867,Z 331.579,A -85,B 0,C 180,E1 -21798.945,E2 -21798.945} C_VEL
LIN {X 0,Y 216.72,Z 341.85,A -85,B 0,C 180,E1 -21800.476,E2 -21800.476} C_VEL
LIN {X 0,Y 212.883,Z 352.311,A -85,B 0,C 180,E1 -21802.433,E2 -21802.433} C_VEL
LIN {X 0,Y 208.925,Z 361.817,A -85,B 0,C 180,E1 -21804.742,E2 -21804.742} C_VEL
LIN {X 0,Y 205.272,Z 369.579,A -85,B 0,C 180,E1 -21807.111,E2 -21807.111} C_VEL
LIN {X 0,Y 201.365,Z 377.469,A -85,B 0,C 180,E1 -21810.227,E2 -21810.227} C_VEL
LIN {X 0,Y 197.943,Z 383.687,A -85,B 0,C 180,E1 -21813.455,E2 -21813.455} C_VEL
LIN {X 0,Y 195.664,Z 387.674,A -85,B 0,C 180,E1 -21816.15,E2 -21816.15} C_VEL
LIN {X 0,Y 193.675,Z 390.896,A -85,B 0,C 180,E1 -21819.021,E2 -21819.021} C_VEL
LIN {X 0,Y 191.767,Z 393.828,A -85,B 0,C 180,E1 -21822.868,E2 -21822.868} C_VEL
LIN {X 0,Y 190.825,Z 395.044,A -85,B 0,C 180,E1 -21825.596,E2 -21825.596} C_VEL
LIN {X 0,Y 190.186,Z 395.586,A -85,B 0,C 180,E1 -21828.309,E2 -21828.309} C_VEL
LIN {X 0,Y 189.794,Z 395.507,A -85,B 0,C 180,E1 -21831.042,E2 -21831.042} C_VEL
LIN {X 0,Y 189.619,Z 394.365,A -85,B 0,C 180,E1 -21834.626,E2 -21834.626} C_VEL
LIN {X 0,Y 189.874,Z 391.914,A -85,B 0,C 180,E1 -21838.354,E2 -21838.354} C_VEL
LIN {X 0,Y 190.65,Z 387.942,A -85,B 0,C 180,E1 -21842.215,E2 -21842.215} C_VEL
LIN {X 0,Y 191.376,Z 384.017,A -85,B 0,C 180,E1 -21845.022,E2 -21845.022} C_VEL
LIN {X 0,Y 192.731,Z 377.542,A -85,B 0,C 180,E1 -21848.616,E2 -21848.616} C_VEL
LIN {X 0,Y 194.269,Z 370.752,A -85,B 0,C 180,E1 -21851.548,E2 -21851.548} C_VEL
LIN {X 0,Y 196.414,Z 361.853,A -85,B 0,C 180,E1 -21854.582,E2 -21854.582} C_VEL
LIN {X 0,Y 198.633,Z 352.097,A -85,B 0,C 180,E1 -21857.227,E2 -21857.227} C_VEL
LIN {X 0,Y 201.108,Z 340.724,A -85,B 0,C 180,E1 -21859.619,E2 -21859.619} C_VEL
LIN {X 0,Y 203.295,Z 328.95,A -85,B 0,C 180,E1 -21861.553,E2 -21861.553} C_VEL
LIN {X 0,Y 205.115,Z 317.305,A -85,B 0,C 180,E1 -21863.01,E2 -21863.01} C_VEL
LIN {X 0,Y 206.746,Z 303.564,A -85,B 0,C 180,E1 -21864.264,E2 -21864.264} C_VEL
LIN {X 0,Y 208.019,Z 290.12,A -85,B 0,C 180,E1 -21865.045,E2 -21865.045} C_VEL
LIN {X 0,Y 210.89,Z 230.421,A -85,B 0,C 180,E1 -21867.222,E2 -21867.222} C_VEL
LIN {X 0,Y 204.268,Z 211.489,A -85,B 0,C 180,E1 -21868.968,E2 -21868.968} C_VEL
LIN {X 0,Y 196.618,Z 192.743,A -85,B 0,C 180,E1 -21871.003,E2 -21871.003} C_VEL
LIN {X 0,Y 193.486,Z 186.876,A -85,B 0,C 180,E1 -21871.849,E2 -21871.849} C_VEL
LIN {X 0,Y 193.223,Z 185.984,A -85,B 0,C 180,E1 -21872.347,E2 -21872.347} C_VEL
LIN {X 0,Y 193.033,Z 185.93,A -85,B 0,C 180,E1 -21878.376,E2 -21878.376} C_VEL
LIN {X 0,Y 192.798,Z 185.956,A -85,B 0,C 180,E1 -21882.636,E2 -21882.636} C_VEL
LIN {X 0,Y 192.757,Z 185.969,A -85,B 0,C 180,E1 -21886.961,E2 -21886.961} C_VEL
LIN {X 0,Y 192.637,Z 185.987,A -85,B 0,C 180,E1 -21891.399,E2 -21891.399} C_VEL
LIN {X 0,Y 192.664,Z 185.978,A -85,B 0,C 180,E1 -21894.227,E2 -21894.227} C_VEL
LIN {X 0,Y 192.645,Z 185.98,A -85,B 0,C 180,E1 -21898.891,E2 -21898.891} C_VEL
LIN {X 0,Y 192.597,Z 185.985,A -85,B 0,C 180,E1 -21903.188,E2 -21903.188} C_VEL
LIN {X 0,Y 192.552,Z 185.983,A -85,B 0,C 180,E1 -21908.354,E2 -21908.354} C_VEL
LIN {X 0,Y 192.494,Z 186.004,A -85,B 0,C 180,E1 -21913.098,E2 -21913.098} C_VEL
LIN {X 0,Y 192.493,Z 185.973,A -85,B 0,C 180,E1 -21916.906,E2 -21916.906} C_VEL
LIN {X 0,Y 192.551,Z 185.983,A -85,B 0,C 180,E1 -21921.649,E2 -21921.649} C_VEL
LIN {X 0,Y 192.597,Z 185.991,A -85,B 0,C 180,E1 -21926.815,E2 -21926.815} C_VEL
LIN {X 0,Y 192.623,Z 185.988,A -85,B 0,C 180,E1 -21931.686,E2 -21931.686} C_VEL
LIN {X 0,Y 192.682,Z 185.971,A -85,B 0,C 180,E1 -21936.347,E2 -21936.347} C_VEL
LIN {X 0,Y 192.736,Z 185.975,A -85,B 0,C 180,E1 -21941.459,E2 -21941.459} C_VEL
LIN {X 0,Y 192.765,Z 185.961,A -85,B 0,C 180,E1 -21945.215,E2 -21945.215} C_VEL
LIN {X 0,Y 192.95,Z 185.949,A -85,B 0,C 180,E1 -21949.568,E2 -21949.568} C_VEL
LIN {X 0,Y 192.968,Z 185.94,A -85,B 0,C 180,E1 -21953.728,E2 -21953.728} C_VEL
LIN {X 0,Y 193.234,Z 185.91,A -85,B 0,C 180,E1 -21957.917,E2 -21957.917} C_VEL
LIN {X 0,Y 193.417,Z 185.874,A -85,B 0,C 180,E1 -21960.001,E2 -21960.001} C_VEL
LIN {X 0,Y 192.94,Z 185.91,A -85,B 0,C 180,E1 -21964.179,E2 -21964.179} C_VEL
LIN {X 0,Y 193.031,Z 185.938,A -85,B 0,C 180,E1 -21968.375,E2 -21968.375} C_VEL
LIN {X 0,Y 192.795,Z 185.96,A -85,B 0,C 180,E1 -21972.635,E2 -21972.635} C_VEL
LIN {X 0,Y 192.717,Z 185.949,A -85,B 0,C 180,E1 -21976.963,E2 -21976.963} C_VEL
LIN {X 0,Y 192.578,Z 185.998,A -85,B 0,C 180,E1 -21981.405,E2 -21981.405} C_VEL
LIN {X 0,Y 192.616,Z 185.977,A -85,B 0,C 180,E1 -21984.189,E2 -21984.189} C_VEL
LIN {X 0,Y 192.606,Z 185.989,A -85,B 0,C 180,E1 -21988.865,E2 -21988.865} C_VEL
LIN {X 0,Y 192.6,Z 185.976,A -85,B 0,C 180,E1 -21993.187,E2 -21993.187} C_VEL
LIN {X 0,Y 192.547,Z 185.996,A -85,B 0,C 180,E1 -21998.354,E2 -21998.354} C_VEL
LIN {X 0,Y 192.49,Z 186.007,A -85,B 0,C 180,E1 -22003.093,E2 -22003.093} C_VEL
LIN {X 0,Y 192.49,Z 186.008,A -85,B 0,C 180,E1 -22006.906,E2 -22006.906} C_VEL
LIN {X 0,Y 192.608,Z 186.148,A -85,B 0,C 180,E1 -22010.021,E2 -22010.021} C_VEL
LIN {X 0,Y 193.505,Z 190.003,A -85,B 0,C 180,E1 -22012.064,E2 -22012.064} C_VEL
LIN {X 0,Y 199.748,Z 204.481,A -85,B 0,C 180,E1 -22013.821,E2 -22013.821} C_VEL
LIN {X 0,Y 206.86,Z 223.066,A -85,B 0,C 180,E1 -22015.692,E2 -22015.692} C_VEL
LIN {X 0,Y 208.786,Z 228.751,A -85,B 0,C 180,E1 -22016.204,E2 -22016.204} C_VEL
LIN {X 0,Y 210.467,Z 243.489,A -85,B 0,C 180,E1 -22017.056,E2 -22017.056} C_VEL
LIN {X 0,Y 209.802,Z 257.738,A -85,B 0,C 180,E1 -22017.569,E2 -22017.569} C_VEL
LIN {X 0,Y 208.942,Z 263.558,A -85,B 0,C 180,E1 -22017.704,E2 -22017.704} C_VEL
LIN {X 0,Y 202.773,Z 282.412,A -85,B 0,C 180,E1 -22017.722,E2 -22017.722} C_VEL
LIN {X 0,Y 201.845,Z 288.233,A -85,B 0,C 180,E1 -22017.856,E2 -22017.856} C_VEL
LIN {X 0,Y 200.953,Z 302.374,A -85,B 0,C 180,E1 -22018.504,E2 -22018.504} C_VEL
LIN {X 0,Y 199.496,Z 314.943,A -85,B 0,C 180,E1 -22019.426,E2 -22019.426} C_VEL
LIN {X 0,Y 197.654,Z 327.31,A -85,B 0,C 180,E1 -22020.729,E2 -22020.729} C_VEL
LIN {X 0,Y 195.444,Z 339.304,A -85,B 0,C 180,E1 -22022.419,E2 -22022.419} C_VEL
LIN {X 0,Y 193.246,Z 350.08,A -85,B 0,C 180,E1 -22024.412,E2 -22024.412} C_VEL
LIN {X 0,Y 190.936,Z 360.189,A -85,B 0,C 180,E1 -22026.769,E2 -22026.769} C_VEL
LIN {X 0,Y 189.316,Z 367.226,A -85,B 0,C 180,E1 -22028.778,E2 -22028.778} C_VEL
LIN {X 0,Y 187.095,Z 376.259,A -85,B 0,C 180,E1 -22031.945,E2 -22031.945} C_VEL
LIN {X 0,Y 185.291,Z 383.479,A -85,B 0,C 180,E1 -22035.164,E2 -22035.164} C_VEL
LIN {X 0,Y 184.006,Z 390.044,A -85,B 0,C 180,E1 -22038.988,E2 -22038.988} C_VEL
LIN {X 0,Y 183.334,Z 394.343,A -85,B 0,C 180,E1 -22042.287,E2 -22042.287} C_VEL
LIN {X 0,Y 183.04,Z 397.532,A -85,B 0,C 180,E1 -22045.594,E2 -22045.594} C_VEL
LIN {X 0,Y 182.999,Z 399.104,A -85,B 0,C 180,E1 -22047.797,E2 -22047.797} C_VEL
LIN {X 0,Y 183.096,Z 400.236,A -85,B 0,C 180,E1 -22049.998,E2 -22049.998} C_VEL
LIN {X 0,Y 183.082,Z 401.227,A -85,B 0,C 180,E1 -22054.401,E2 -22054.401} C_VEL
LIN {X 0,Y 183.301,Z 401.146,A -85,B 0,C 180,E1 -22056.603,E2 -22056.603} C_VEL
LIN {X 0,Y 183.636,Z 400.671,A -85,B 0,C 180,E1 -22058.803,E2 -22058.803} C_VEL
LIN {X 0,Y 185.026,Z 398.485,A -85,B 0,C 180,E1 -22063.171,E2 -22063.171} C_VEL
LIN {X 0,Y 186.641,Z 395.787,A -85,B 0,C 180,E1 -22066.402,E2 -22066.402} C_VEL
LIN {X 0,Y 188.942,Z 392.097,A -85,B 0,C 180,E1 -22069.556,E2 -22069.556} C_VEL
LIN {X 0,Y 191.934,Z 387.331,A -85,B 0,C 180,E1 -22072.608,E2 -22072.608} C_VEL
